C05446=1127.597,405.977,-90.668,-176.772,11.513,149.514
C05447=1127.600,405.729,-90.630,-176.772,11.509,149.513
C05448=1127.605,405.482,-90.592,-176.773,11.506,149.513
C05449=1127.608,405.235,-90.554,-176.773,11.502,149.512
C05450=1127.611,404.988,-90.515,-176.773,11.498,149.511
C05451=1127.615,404.742,-90.477,-176.773,11.494,149.510
C05452=1127.619,404.494,-90.439,-176.774,11.491,149.509
C05453=1127.622,404.247,-90.401,-176.773,11.488,149.508
C05454=1127.626,404.000,-90.362,-176.774,11.484,149.507
C05455=1127.630,403.753,-90.324,-176.774,11.481,149.506
C05456=1127.633,403.541,-90.291,-176.774,11.477,149.505
C05457=1127.637,403.328,-90.259,-176.774,11.474,149.505
C05458=1127.639,403.116,-90.225,-176.774,11.472,149.504
C05459=1127.643,402.904,-90.192,-176.775,11.468,149.503
C05460=1127.646,402.691,-90.160,-176.775,11.466,149.503
C05461=1127.649,402.480,-90.127,-176.775,11.462,149.502
C05462=1127.651,402.267,-90.094,-176.775,11.460,149.501
C05463=1127.655,402.055,-90.062,-176.776,11.457,149.501
C05464=1127.659,401.808,-90.023,-176.776,11.454,149.500
C05465=1127.662,401.561,-89.985,-176.777,11.450,149.499
C05466=1127.666,401.314,-89.947,-176.777,11.447,149.498
C05467=1127.670,401.067,-89.909,-176.778,11.443,149.498
C05468=1127.673,400.820,-89.871,-176.778,11.441,149.497
C05469=1127.677,400.572,-89.832,-176.778,11.437,149.496
C05470=1127.681,400.325,-89.795,-176.779,11.434,149.495
C05471=1127.684,400.078,-89.757,-176.779,11.431,149.495
C05472=1127.688,399.832,-89.718,-176.780,11.428,149.494
C05473=1127.692,399.585,-89.680,-176.781,11.425,149.493
C05474=1127.695,399.337,-89.641,-176.781,11.422,149.493
C05475=1127.699,399.091,-89.604,-176.781,11.419,149.492
C05476=1127.702,398.843,-89.566,-176.782,11.415,149.491
C05477=1127.707,398.596,-89.528,-176.782,11.413,149.491
C05478=1127.710,398.349,-89.490,-176.783,11.410,149.490
C05479=1127.714,398.102,-89.451,-176.784,11.407,149.490
C05480=1127.718,397.855,-89.414,-176.784,11.404,149.489
C05481=1127.721,397.608,-89.376,-176.785,11.401,149.488
C05482=1127.726,397.361,-89.338,-176.786,11.398,149.488
C05483=1127.729,397.114,-89.300,-176.787,11.396,149.487
C05484=1127.733,396.867,-89.262,-176.787,11.392,149.487
C05485=1127.736,396.619,-89.223,-176.788,11.389,149.486
C05486=1127.740,396.372,-89.186,-176.789,11.387,149.486
C05487=1127.743,396.126,-89.148,-176.790,11.384,149.485
C05488=1127.747,395.878,-89.109,-176.790,11.382,149.485
C05489=1127.751,395.631,-89.072,-176.791,11.379,149.484
C05490=1127.754,395.384,-89.034,-176.792,11.376,149.484
C05491=1127.759,395.137,-88.996,-176.793,11.373,149.483
C05492=1127.762,394.890,-88.958,-176.794,11.370,149.483
C05493=1127.766,394.643,-88.920,-176.795,11.368,149.482
C05494=1127.770,394.396,-88.882,-176.796,11.365,149.482
C05495=1127.773,394.149,-88.844,-176.796,11.363,149.481
C05496=1127.777,393.902,-88.806,-176.797,11.360,149.481
C05497=1127.780,393.655,-88.768,-176.798,11.358,149.481
C05498=1127.784,393.408,-88.730,-176.799,11.355,149.480
C05499=1127.788,393.161,-88.692,-176.800,11.353,149.480
C05500=1127.791,392.914,-88.655,-176.801,11.350,149.479
C05501=1127.796,392.666,-88.617,-176.802,11.348,149.479
C05502=1127.799,392.419,-88.579,-176.803,11.345,149.479
C05503=1127.803,392.172,-88.541,-176.804,11.343,149.478
C05504=1127.806,391.925,-88.504,-176.805,11.340,149.478
C05505=1127.810,391.678,-88.466,-176.806,11.339,149.477
C05506=1127.814,391.431,-88.428,-176.807,11.336,149.477
C05507=1127.817,391.184,-88.390,-176.808,11.334,149.477
C05508=1127.821,390.937,-88.352,-176.810,11.331,149.477
C05509=1127.825,390.689,-88.315,-176.811,11.329,149.476
C05510=1127.829,390.443,-88.277,-176.811,11.327,149.476
C05511=1127.832,390.195,-88.239,-176.813,11.325,149.476
C05512=1127.836,389.983,-88.206,-176.814,11.323,149.475
C05513=1127.839,389.771,-88.174,-176.815,11.321,149.475
C05514=1127.842,389.559,-88.142,-176.815,11.319,149.475
C05515=1127.845,389.346,-88.109,-176.817,11.318,149.475
C05516=1127.848,389.134,-88.077,-176.818,11.316,149.475
C05517=1127.851,388.921,-88.044,-176.818,11.314,149.474
C05518=1127.855,388.709,-88.011,-176.820,11.312,149.474
C05519=1127.857,388.497,-87.979,-176.821,11.309,149.474
C05520=1127.862,388.249,-87.942,-176.822,11.308,149.474
C05521=1127.865,388.002,-87.904,-176.823,11.306,149.473
C05522=1127.869,387.755,-87.866,-176.825,11.304,149.473
C05523=1127.872,387.508,-87.829,-176.826,11.302,149.473
C05524=1127.876,387.260,-87.791,-176.827,11.300,149.473
C05525=1127.880,387.014,-87.754,-176.829,11.297,149.473
C05526=1127.884,386.766,-87.715,-176.830,11.296,149.473
C05527=1127.888,386.519,-87.678,-176.832,11.294,149.472
C05528=1127.891,386.272,-87.640,-176.833,11.292,149.472
C05529=1127.895,386.025,-87.603,-176.834,11.290,149.472
C05530=1127.898,385.779,-87.565,-176.836,11.288,149.472
C05531=1127.902,385.531,-87.528,-176.837,11.286,149.472
C05532=1127.906,385.284,-87.490,-176.838,11.285,149.472
C05533=1127.909,385.037,-87.452,-176.840,11.282,149.472
C05534=1127.914,384.789,-87.415,-176.841,11.281,149.472
C05535=1127.917,384.542,-87.377,-176.843,11.279,149.471
C05536=1127.921,384.295,-87.340,-176.845,11.277,149.471
C05537=1127.924,384.048,-87.302,-176.846,11.275,149.471
C05538=1127.928,383.801,-87.265,-176.847,11.274,149.471
C05539=1127.932,383.554,-87.228,-176.849,11.271,149.471
C05540=1127.935,383.307,-87.190,-176.851,11.269,149.471
C05541=1127.939,383.060,-87.152,-176.853,11.267,149.471
C05542=1127.943,382.812,-87.115,-176.856,11.264,149.471
C05543=1127.946,382.566,-87.078,-176.859,11.262,149.471
C05544=1127.951,382.318,-87.040,-176.862,11.260,149.471
C05545=1127.954,382.071,-87.002,-176.865,11.257,149.471
C05546=1127.958,381.824,-86.965,-176.867,11.255,149.471
C05547=1127.962,381.576,-86.927,-176.870,11.252,149.472
C05548=1127.966,381.329,-86.891,-176.873,11.250,149.472
C05549=1127.969,381.083,-86.853,-176.876,11.248,149.472
C05550=1127.973,380.835,-86.816,-176.878,11.246,149.472
C05551=1127.977,380.588,-86.778,-176.881,11.243,149.472
C05552=1127.980,380.340,-86.741,-176.884,11.240,149.472
C05553=1127.984,380.094,-86.703,-176.887,11.239,149.472
C05554=1127.988,379.846,-86.666,-176.890,11.236,149.472
C05555=1127.992,379.599,-86.629,-176.892,11.233,149.472
C05556=1127.995,379.352,-86.592,-176.895,11.231,149.472
C05557=1128.000,379.105,-86.555,-176.898,11.228,149.472
C05558=1128.003,378.858,-86.517,-176.901,11.227,149.473
C05559=1128.007,378.610,-86.480,-176.904,11.224,149.473
C05560=1128.011,378.363,-86.443,-176.907,11.221,149.473
C05561=1128.013,378.116,-86.406,-176.909,11.219,149.473
C05562=1128.017,377.869,-86.369,-176.912,11.217,149.473
C05563=1128.022,377.622,-86.332,-176.915,11.214,149.473
C05564=1128.025,377.374,-86.295,-176.918,11.212,149.473
C05565=1128.029,377.127,-86.257,-176.921,11.210,149.474
C05566=1128.033,376.880,-86.220,-176.924,11.208,149.474
C05567=1128.037,376.633,-86.184,-176.927,11.205,149.474
C05568=1128.040,376.421,-86.152,-176.929,11.203,149.474
C05569=1128.044,376.208,-86.120,-176.932,11.202,149.474
C05570=1128.046,375.996,-86.088,-176.935,11.199,149.474
C05571=1128.050,375.783,-86.056,-176.937,11.197,149.474
C05572=1128.053,375.570,-86.025,-176.940,11.195,149.475
C05573=1128.056,375.358,-85.993,-176.942,11.193,149.475
C05574=1128.060,375.145,-85.961,-176.945,11.191,149.475
C05575=1128.062,374.933,-85.929,-176.947,11.189,149.475
C05576=1128.066,374.685,-85.892,-176.950,11.187,149.475
C05577=1128.070,374.438,-85.855,-176.954,11.184,149.475
C05578=1128.074,374.191,-85.818,-176.956,11.183,149.476
C05579=1128.077,373.944,-85.782,-176.959,11.180,149.476
C05580=1128.081,373.696,-85.744,-176.962,11.178,149.476
C05581=1128.085,373.449,-85.707,-176.966,11.175,149.476
C05582=1128.089,373.202,-85.671,-176.968,11.173,149.476
C05583=1128.093,372.955,-85.634,-176.972,11.171,149.476
C05584=1128.097,372.708,-85.597,-176.975,11.168,149.477
C05585=1128.100,372.460,-85.560,-176.977,11.166,149.477
C05586=1128.104,372.213,-85.523,-176.981,11.164,149.477
C05587=1128.107,371.966,-85.487,-176.984,11.161,149.477
C05588=1128.112,371.719,-85.450,-176.987,11.159,149.477
C05589=1128.116,371.471,-85.413,-176.990,11.157,149.478
C05590=1128.119,371.224,-85.376,-176.993,11.155,149.478
C05591=1128.123,370.977,-85.340,-176.996,11.152,149.478
C05592=1128.127,370.729,-85.303,-177.000,11.150,149.478
C05593=1128.131,370.482,-85.266,-177.002,11.148,149.478
C05594=1128.134,370.235,-85.230,-177.006,11.146,149.479
C05595=1128.138,369.988,-85.193,-177.009,11.143,149.479
C05596=1128.142,369.740,-85.156,-177.012,11.141,149.479
C05597=1128.145,369.493,-85.120,-177.016,11.138,149.479
C05598=1128.149,369.246,-85.083,-177.018,11.137,149.480
C05599=1128.154,368.998,-85.047,-177.022,11.134,149.480
C05600=1128.157,368.752,-85.010,-177.025,11.132,149.480
C05601=1128.161,368.504,-84.973,-177.028,11.129,149.480
C05602=1128.164,368.258,-84.937,-177.031,11.127,149.480
C05603=1128.168,368.009,-84.901,-177.034,11.125,149.481
C05604=1128.172,367.762,-84.864,-177.037,11.122,149.481
C05605=1128.176,367.515,-84.828,-177.041,11.120,149.481
C05606=1128.180,367.267,-84.791,-177.044,11.117,149.481
C05607=1128.183,367.020,-84.755,-177.047,11.115,149.481
C05608=1128.187,366.773,-84.718,-177.051,11.113,149.482
C05609=1128.191,366.526,-84.682,-177.054,11.110,149.482
C05610=1128.195,366.278,-84.646,-177.057,11.108,149.482
C05611=1128.199,366.031,-84.610,-177.060,11.106,149.483
C05612=1128.203,365.784,-84.573,-177.064,11.104,149.483
C05613=1128.207,365.536,-84.537,-177.067,11.101,149.483
C05614=1128.210,365.289,-84.500,-177.070,11.099,149.483
C05615=1128.214,365.041,-84.464,-177.073,11.096,149.483
C05616=1128.218,364.794,-84.428,-177.077,11.094,149.484
C05617=1128.221,364.547,-84.392,-177.080,11.091,149.484
C05618=1128.225,364.299,-84.355,-177.084,11.089,149.484
C05619=1128.229,364.053,-84.319,-177.086,11.088,149.484
C05620=1128.233,363.805,-84.283,-177.090,11.085,149.485
C05621=1128.236,363.558,-84.247,-177.093,11.083,149.485
C05622=1128.241,363.310,-84.210,-177.096,11.080,149.485
C05623=1128.244,363.063,-84.174,-177.100,11.078,149.485
C05624=1128.248,362.850,-84.144,-177.103,11.075,149.486
C05625=1128.251,362.637,-84.112,-177.106,11.074,149.486
C05626=1128.254,362.425,-84.081,-177.108,11.072,149.486
C05627=1128.257,362.213,-84.050,-177.112,11.069,149.486
C05628=1128.261,361.999,-84.020,-177.114,11.068,149.486
C05629=1128.264,361.787,-83.988,-177.118,11.065,149.487
C05630=1128.267,361.575,-83.957,-177.120,11.064,149.487
C05631=1128.271,361.362,-83.927,-177.124,11.061,149.487
C05632=1128.274,361.115,-83.891,-177.127,11.059,149.487
C05633=1128.278,360.867,-83.854,-177.130,11.056,149.488
C05634=1128.282,360.619,-83.819,-177.134,11.054,149.488
C05635=1128.285,360.372,-83.783,-177.137,11.052,149.488
C05636=1128.290,360.125,-83.746,-177.141,11.049,149.488
C05637=1128.293,359.877,-83.711,-177.144,11.047,149.489
C05638=1128.297,359.630,-83.675,-177.147,11.044,149.489
C05639=1128.301,359.382,-83.638,-177.151,11.042,149.489
C05640=1128.305,359.135,-83.603,-177.154,11.039,149.490
C05641=1128.309,358.887,-83.567,-177.157,11.037,149.490
C05642=1128.312,358.641,-83.531,-177.161,11.035,149.490
C05643=1128.316,358.393,-83.495,-177.164,11.032,149.490
C05644=1128.321,358.146,-83.460,-177.168,11.030,149.491
C05645=1128.324,357.898,-83.424,-177.171,11.027,149.491
C05646=1128.328,357.651,-83.389,-177.174,11.025,149.491
C05647=1128.332,357.403,-83.353,-177.178,11.023,149.491
C05648=1128.336,357.156,-83.317,-177.182,11.020,149.492
C05649=1128.339,356.909,-83.281,-177.185,11.017,149.492
C05650=1128.343,356.661,-83.245,-177.189,11.015,149.492
C05651=1128.347,356.414,-83.210,-177.192,11.013,149.492
C05652=1128.350,356.166,-83.174,-177.196,11.010,149.493
C05653=1128.355,355.920,-83.139,-177.199,11.008,149.493
C05654=1128.359,355.672,-83.103,-177.203,11.005,149.493
C05655=1128.363,355.424,-83.067,-177.207,11.002,149.493
C05656=1128.366,355.177,-83.032,-177.210,11.000,149.494
C05657=1128.370,354.929,-82.996,-177.213,10.997,149.494
C05658=1128.374,354.682,-82.961,-177.217,10.995,149.494
C05659=1128.378,354.435,-82.925,-177.221,10.992,149.495
C05660=1128.382,354.187,-82.890,-177.224,10.989,149.495
C05661=1128.385,353.940,-82.854,-177.228,10.987,149.495
C05662=1128.389,353.692,-82.819,-177.231,10.985,149.495
C05663=1128.394,353.444,-82.783,-177.235,10.982,149.496
C05664=1128.398,353.197,-82.748,-177.238,10.979,149.496
C05665=1128.402,352.950,-82.713,-177.242,10.977,149.496
C05666=1128.405,352.702,-82.677,-177.245,10.975,149.496
C05667=1128.409,352.455,-82.642,-177.249,10.971,149.497
C05668=1128.413,352.208,-82.606,-177.253,10.969,149.497
C05669=1128.417,351.960,-82.571,-177.256,10.966,149.497
C05670=1128.421,351.712,-82.536,-177.260,10.964,149.497
C05671=1128.424,351.465,-82.500,-177.264,10.961,149.498
C05672=1128.429,351.218,-82.465,-177.267,10.959,149.498
C05673=1128.433,350.970,-82.430,-177.271,10.955,149.498
C05674=1128.436,350.722,-82.395,-177.275,10.953,149.498
C05675=1128.440,350.475,-82.359,-177.278,10.951,149.499
C05676=1128.444,350.228,-82.325,-177.282,10.948,149.499
C05677=1128.447,349.980,-82.290,-177.285,10.945,149.499
C05678=1128.451,349.733,-82.254,-177.289,10.943,149.500
C05679=1128.456,349.485,-82.220,-177.293,10.940,149.500
C05680=1128.459,349.272,-82.189,-177.295,10.938,149.500
C05681=1128.463,349.059,-82.159,-177.298,10.935,149.500
C05682=1128.466,348.846,-82.129,-177.301,10.934,149.500
C05683=1128.469,348.633,-82.099,-177.303,10.932,149.500
C05684=1128.472,348.421,-82.069,-177.307,10.929,149.501
C05685=1128.476,348.208,-82.038,-177.309,10.927,149.501
C05686=1128.479,347.995,-82.008,-177.312,10.925,149.501
C05687=1128.482,347.782,-81.978,-177.315,10.923,149.501
C05688=1128.486,347.535,-81.943,-177.318,10.920,149.501
C05689=1128.490,347.287,-81.908,-177.321,10.918,149.501
C05690=1128.494,347.040,-81.873,-177.325,10.915,149.502
C05691=1128.499,346.792,-81.838,-177.328,10.913,149.502
C05692=1128.502,346.544,-81.804,-177.331,10.910,149.502
C05693=1128.506,346.298,-81.769,-177.335,10.908,149.502
C05694=1128.510,346.050,-81.734,-177.338,10.905,149.503
C05695=1128.514,345.802,-81.698,-177.341,10.903,149.503
C05696=1128.518,345.555,-81.664,-177.344,10.900,149.503
C05697=1128.521,345.307,-81.630,-177.347,10.898,149.503
C05698=1128.526,345.060,-81.595,-177.351,10.895,149.503
C05699=1128.530,344.812,-81.560,-177.354,10.893,149.504
C05700=1128.534,344.564,-81.525,-177.357,10.890,149.504
C05701=1128.537,344.317,-81.490,-177.360,10.889,149.504
C05702=1128.541,344.069,-81.455,-177.363,10.886,149.504
C05703=1128.546,343.822,-81.421,-177.366,10.883,149.504
C05704=1128.549,343.575,-81.386,-177.370,10.881,149.505
C05705=1128.553,343.327,-81.352,-177.373,10.878,149.505
C05706=1128.557,343.079,-81.317,-177.376,10.876,149.505
C05707=1128.562,342.832,-81.282,-177.379,10.874,149.505
C05708=1128.565,342.584,-81.247,-177.383,10.871,149.506
C05709=1128.569,342.336,-81.212,-177.386,10.868,149.506
C05710=1128.573,342.089,-81.178,-177.389,10.866,149.506
C05711=1128.576,341.841,-81.144,-177.392,10.863,149.506
C05712=1128.581,341.594,-81.109,-177.396,10.861,149.506
C05713=1128.584,341.346,-81.075,-177.399,10.859,149.507
C05714=1128.589,341.099,-81.040,-177.402,10.856,149.507
C05715=1128.593,340.851,-81.005,-177.405,10.853,149.507
C05716=1128.596,340.604,-80.971,-177.409,10.851,149.507
C05717=1128.601,340.356,-80.937,-177.412,10.848,149.507
C05718=1128.605,340.108,-80.902,-177.415,10.846,149.507
C05719=1128.609,339.861,-80.868,-177.418,10.843,149.508
C05720=1128.613,339.613,-80.833,-177.421,10.841,149.508
C05721=1128.617,339.366,-80.799,-177.425,10.838,149.508
C05722=1128.620,339.118,-80.764,-177.428,10.836,149.508
C05723=1128.624,338.871,-80.731,-177.431,10.833,149.508
C05724=1128.628,338.623,-80.696,-177.434,10.831,149.509
C05725=1128.632,338.375,-80.662,-177.438,10.828,149.509
C05726=1128.636,338.127,-80.627,-177.440,10.826,149.509
C05727=1128.640,337.880,-80.593,-177.444,10.824,149.509
C05728=1128.644,337.633,-80.559,-177.447,10.822,149.510
C05729=1128.648,337.385,-80.525,-177.450,10.819,149.510
C05730=1128.652,337.138,-80.490,-177.453,10.816,149.510
C05731=1128.656,336.890,-80.456,-177.456,10.814,149.510
C05732=1128.660,336.642,-80.422,-177.460,10.811,149.510
C05733=1128.664,336.394,-80.388,-177.463,10.809,149.511
C05734=1128.668,336.147,-80.353,-177.466,10.806,149.511
C05735=1128.672,335.899,-80.319,-177.469,10.804,149.511
C05736=1128.675,335.686,-80.290,-177.472,10.802,149.511
C05737=1128.679,335.473,-80.260,-177.475,10.799,149.511
C05738=1128.682,335.260,-80.231,-177.478,10.798,149.511
C05739=1128.685,335.047,-80.202,-177.481,10.795,149.511
C05740=1128.689,334.834,-80.173,-177.483,10.793,149.512
C05741=1128.692,334.622,-80.143,-177.486,10.790,149.512
C05742=1128.696,334.409,-80.115,-177.489,10.789,149.512
C05743=1128.699,334.195,-80.085,-177.491,10.787,149.512
C05744=1128.703,333.948,-80.051,-177.494,10.784,149.512
C05745=1128.707,333.701,-80.017,-177.498,10.782,149.513
C05746=1128.711,333.452,-79.983,-177.501,10.779,149.513
C05747=1128.715,333.205,-79.949,-177.504,10.776,149.513
C05748=1128.719,332.958,-79.915,-177.507,10.774,149.513
C05749=1128.723,332.709,-79.881,-177.511,10.772,149.513
C05750=1128.727,332.462,-79.847,-177.514,10.769,149.513
C05751=1128.731,332.214,-79.814,-177.517,10.766,149.514
C05752=1128.735,331.966,-79.779,-177.520,10.764,149.514
C05753=1128.739,331.719,-79.745,-177.524,10.761,149.514
C05754=1128.743,331.471,-79.712,-177.526,10.759,149.514
C05755=1128.746,331.223,-79.678,-177.530,10.756,149.514
C05756=1128.751,330.975,-79.644,-177.533,10.754,149.515
C05757=1128.755,330.728,-79.610,-177.536,10.751,149.515
C05758=1128.759,330.480,-79.577,-177.539,10.749,149.515
C05759=1128.762,330.233,-79.543,-177.543,10.746,149.515
C05760=1128.766,329.985,-79.510,-177.546,10.744,149.516
C05761=1128.771,329.737,-79.475,-177.548,10.742,149.516
C05762=1128.775,329.489,-79.442,-177.552,10.739,149.516
C05763=1128.778,329.242,-79.408,-177.555,10.737,149.516
C05764=1128.783,328.994,-79.375,-177.558,10.734,149.516
C05765=1128.786,328.747,-79.341,-177.561,10.732,149.516
C05766=1128.791,328.498,-79.307,-177.564,10.729,149.517
C05767=1128.795,328.251,-79.274,-177.568,10.727,149.517
C05768=1128.799,328.004,-79.240,-177.571,10.724,149.517
C05769=1128.803,327.756,-79.206,-177.574,10.721,149.517
C05770=1128.807,327.508,-79.173,-177.577,10.719,149.517
C05771=1128.810,327.260,-79.139,-177.581,10.717,149.518
C05772=1128.814,327.013,-79.106,-177.584,10.714,149.518
C05773=1128.818,326.765,-79.073,-177.587,10.711,149.518
C05774=1128.823,326.517,-79.038,-177.590,10.709,149.518
C05775=1128.827,326.270,-79.005,-177.593,10.706,149.518
C05776=1128.831,326.021,-78.972,-177.597,10.704,149.519
C05777=1128.835,325.773,-78.938,-177.600,10.701,149.519
C05778=1128.839,325.526,-78.905,-177.603,10.698,149.519
C05779=1128.843,325.279,-78.871,-177.606,10.696,149.519
C05780=1128.847,325.031,-78.838,-177.609,10.694,149.519
C05781=1128.851,324.783,-78.805,-177.612,10.691,149.519
C05782=1128.855,324.535,-78.772,-177.615,10.689,149.520
C05783=1128.858,324.288,-78.738,-177.618,10.687,149.520
C05784=1128.863,324.040,-78.705,-177.622,10.684,149.520
C05785=1128.867,323.792,-78.671,-177.625,10.681,149.520
C05786=1128.871,323.544,-78.638,-177.628,10.679,149.521
C05787=1128.875,323.297,-78.605,-177.631,10.677,149.521
C05788=1128.879,323.049,-78.572,-177.634,10.674,149.521
C05789=1128.883,322.801,-78.539,-177.637,10.671,149.521
C05790=1128.887,322.553,-78.505,-177.641,10.669,149.521
C05791=1128.891,322.305,-78.472,-177.644,10.666,149.521
C05792=1128.894,322.093,-78.444,-177.646,10.664,149.522
C05793=1128.898,321.879,-78.416,-177.649,10.662,149.522
C05794=1128.901,321.666,-78.387,-177.652,10.660,149.522
C05795=1128.905,321.453,-78.358,-177.655,10.657,149.522
C05796=1128.908,321.240,-78.330,-177.657,10.655,149.522
C05797=1128.911,321.027,-78.301,-177.660,10.654,149.522
C05798=1128.915,320.814,-78.273,-177.663,10.651,149.523
C05799=1128.919,320.601,-78.244,-177.666,10.649,149.523
C05800=1128.923,320.353,-78.211,-177.669,10.646,149.523
C05801=1128.927,320.105,-78.178,-177.672,10.644,149.523
C05802=1128.930,319.857,-78.145,-177.675,10.641,149.523
C05803=1128.934,319.610,-78.112,-177.678,10.639,149.523
C05804=1128.938,319.361,-78.080,-177.681,10.636,149.524
C05805=1128.942,319.113,-78.046,-177.684,10.633,149.524
C05806=1128.946,318.866,-78.013,-177.688,10.631,149.524
C05807=1128.950,318.618,-77.981,-177.691,10.629,149.524
C05808=1128.954,318.371,-77.948,-177.694,10.626,149.524
C05809=1128.958,318.123,-77.914,-177.697,10.623,149.525
C05810=1128.963,317.874,-77.882,-177.701,10.621,149.525
C05811=1128.967,317.627,-77.849,-177.703,10.619,149.525
C05812=1128.970,317.379,-77.816,-177.706,10.617,149.525
C05813=1128.974,317.132,-77.783,-177.710,10.614,149.525
C05814=1128.979,316.883,-77.751,-177.712,10.611,149.526
C05815=1128.983,316.636,-77.717,-177.716,10.609,149.526
C05816=1128.986,316.388,-77.685,-177.719,10.606,149.526
C05817=1128.991,316.140,-77.652,-177.722,10.604,149.526
C05818=1128.995,315.892,-77.619,-177.725,10.601,149.526
C05819=1128.998,315.645,-77.587,-177.728,10.598,149.526
C05820=1129.003,315.396,-77.554,-177.732,10.596,149.527
C05821=1129.007,315.149,-77.522,-177.735,10.593,149.527
C05822=1129.011,314.902,-77.489,-177.738,10.591,149.527
C05823=1129.015,314.653,-77.457,-177.741,10.588,149.527
C05824=1129.019,314.406,-77.423,-177.744,10.586,149.527
C05825=1129.023,314.158,-77.392,-177.747,10.583,149.528
C05826=1129.027,313.910,-77.358,-177.750,10.580,149.528
C05827=1129.031,313.662,-77.325,-177.754,10.578,149.528
C05828=1129.035,313.414,-77.293,-177.757,10.575,149.528
C05829=1129.039,313.166,-77.260,-177.759,10.573,149.528
C05830=1129.043,312.918,-77.228,-177.763,10.571,149.529
C05831=1129.047,312.671,-77.195,-177.766,10.568,149.529
C05832=1129.052,312.422,-77.163,-177.769,10.566,149.529
C05833=1129.056,312.176,-77.131,-177.772,10.563,149.529
C05834=1129.060,311.927,-77.098,-177.775,10.561,149.529
C05835=1129.064,311.679,-77.066,-177.779,10.558,149.529
C05836=1129.068,311.432,-77.033,-177.781,10.555,149.530
C05837=1129.072,311.183,-77.001,-177.785,10.553,149.530
C05838=1129.076,310.936,-76.968,-177.788,10.551,149.530
C05839=1129.079,310.688,-76.936,-177.791,10.548,149.530
C05840=1129.084,310.440,-76.904,-177.794,10.545,149.530
C05841=1129.088,310.193,-76.872,-177.797,10.543,149.530
C05842=1129.092,309.944,-76.839,-177.801,10.540,149.531
C05843=1129.096,309.696,-76.807,-177.804,10.537,149.531
C05844=1129.100,309.449,-76.774,-177.807,10.535,149.531
C05845=1129.104,309.200,-76.742,-177.810,10.533,149.531
C05846=1129.109,308.953,-76.710,-177.813,10.531,149.531
C05847=1129.113,308.705,-76.678,-177.816,10.528,149.532
C05848=1129.116,308.491,-76.650,-177.819,10.525,149.532
C05849=1129.119,308.278,-76.623,-177.821,10.523,149.532
C05850=1129.123,308.065,-76.595,-177.824,10.522,149.532
C05851=1129.126,307.851,-76.567,-177.827,10.519,149.532
C05852=1129.130,307.639,-76.540,-177.829,10.517,149.533
C05853=1129.134,307.425,-76.512,-177.832,10.514,149.533
C05854=1129.137,307.212,-76.484,-177.835,10.512,149.533
C05855=1129.141,306.998,-76.457,-177.837,10.511,149.533
C05856=1129.145,306.751,-76.424,-177.840,10.508,149.533
C05857=1129.149,306.503,-76.393,-177.844,10.506,149.533
C05858=1129.153,306.255,-76.360,-177.847,10.503,149.533
C05859=1129.157,306.007,-76.328,-177.850,10.500,149.534
C05860=1129.161,305.759,-76.296,-177.853,10.498,149.534
C05861=1129.166,305.511,-76.264,-177.856,10.495,149.534
C05862=1129.169,305.263,-76.232,-177.859,10.492,149.534
C05863=1129.174,305.015,-76.200,-177.862,10.490,149.534
C05864=1129.178,304.768,-76.169,-177.865,10.487,149.534
C05865=1129.182,304.519,-76.137,-177.869,10.485,149.535
C05866=1129.186,304.271,-76.105,-177.872,10.482,149.535
C05867=1129.190,304.023,-76.072,-177.875,10.480,149.535
C05868=1129.194,303.776,-76.041,-177.878,10.478,149.535
C05869=1129.198,303.528,-76.009,-177.881,10.475,149.535
C05870=1129.203,303.279,-75.977,-177.884,10.473,149.536
C05871=1129.207,303.032,-75.945,-177.887,10.470,149.536
C05872=1129.211,302.784,-75.913,-177.890,10.468,149.536
C05873=1129.214,302.536,-75.881,-177.893,10.465,149.536
C05874=1129.219,302.288,-75.849,-177.896,10.462,149.536
C05875=1129.223,302.040,-75.818,-177.899,10.460,149.536
C05876=1129.227,301.793,-75.786,-177.903,10.457,149.537
C05877=1129.231,301.544,-75.755,-177.906,10.454,149.537
C05878=1129.235,301.296,-75.723,-177.909,10.452,149.537
C05879=1129.240,301.049,-75.691,-177.912,10.449,149.537
C05880=1129.244,300.801,-75.659,-177.915,10.447,149.537
C05881=1129.247,300.552,-75.627,-177.919,10.444,149.538
C05882=1129.252,300.305,-75.597,-177.921,10.442,149.538
C05883=1129.256,300.056,-75.565,-177.924,10.440,149.538
C05884=1129.260,299.809,-75.533,-177.927,10.437,149.538
C05885=1129.265,299.561,-75.501,-177.930,10.435,149.538
C05886=1129.269,299.312,-75.470,-177.933,10.432,149.538
C05887=1129.273,299.065,-75.438,-177.937,10.430,149.539
C05888=1129.277,298.817,-75.406,-177.940,10.427,149.539
C05889=1129.281,298.569,-75.376,-177.943,10.424,149.539
C05890=1129.285,298.321,-75.344,-177.946,10.422,149.539
C05891=1129.289,298.073,-75.312,-177.949,10.419,149.539
C05892=1129.293,297.825,-75.281,-177.952,10.416,149.540
C05893=1129.297,297.577,-75.249,-177.956,10.414,149.540
C05894=1129.301,297.329,-75.218,-177.958,10.411,149.540
C05895=1129.305,297.081,-75.187,-177.961,10.410,149.540
C05896=1129.310,296.833,-75.155,-177.964,10.407,149.540
C05897=1129.314,296.585,-75.124,-177.967,10.404,149.541
C05898=1129.318,296.337,-75.093,-177.970,10.402,149.541
C05899=1129.322,296.089,-75.060,-177.974,10.399,149.541
C05900=1129.326,295.841,-75.030,-177.977,10.396,149.541
C05901=1129.330,295.593,-74.998,-177.980,10.394,149.541
C05902=1129.334,295.345,-74.967,-177.983,10.391,149.541
C05903=1129.338,295.097,-74.936,-177.986,10.389,149.542
C05904=1129.342,294.884,-74.909,-177.989,10.387,149.542
C05905=1129.346,294.670,-74.882,-177.991,10.384,149.542
C05906=1129.349,294.457,-74.855,-177.994,10.382,149.542
C05907=1129.352,294.243,-74.828,-177.996,10.380,149.542
C05908=1129.356,294.030,-74.801,-177.999,10.378,149.542
C05909=1129.359,293.817,-74.774,-178.002,10.376,149.542
C05910=1129.363,293.603,-74.748,-178.004,10.374,149.543
C05911=1129.367,293.390,-74.721,-178.007,10.371,149.543
C05912=1129.371,293.142,-74.689,-178.010,10.368,149.543
C05913=1129.375,292.894,-74.658,-178.014,10.366,149.543
C05914=1129.380,292.646,-74.628,-178.017,10.363,149.543
C05915=1129.384,292.398,-74.596,-178.019,10.362,149.544
C05916=1129.388,292.150,-74.565,-178.022,10.359,149.544
C05917=1129.391,291.901,-74.535,-178.026,10.356,149.544
C05918=1129.396,291.653,-74.504,-178.028,10.354,149.544
C05919=1129.400,291.405,-74.472,-178.032,10.351,149.544
C05920=1129.404,291.157,-74.441,-178.035,10.348,149.544
C05921=1129.408,290.909,-74.410,-178.038,10.346,149.544
C05922=1129.413,290.661,-74.379,-178.041,10.343,149.545
C05923=1129.417,290.414,-74.348,-178.044,10.341,149.545
C05924=1129.421,290.165,-74.317,-178.047,10.338,149.545
C05925=1129.425,289.917,-74.286,-178.050,10.335,149.545
C05926=1129.429,289.668,-74.255,-178.054,10.333,149.545
C05927=1129.433,289.421,-74.224,-178.056,10.331,149.546
C05928=1129.437,289.173,-74.194,-178.059,10.329,149.546
C05929=1129.441,288.925,-74.163,-178.062,10.326,149.546
C05930=1129.446,288.677,-74.132,-178.066,10.323,149.546
C05931=1129.450,288.429,-74.102,-178.068,10.321,149.546
C05932=1129.454,288.180,-74.071,-178.071,10.318,149.546
C05933=1129.458,287.933,-74.040,-178.075,10.315,149.547
C05934=1129.463,287.685,-74.009,-178.078,10.313,149.547
C05935=1129.466,287.436,-73.978,-178.081,10.310,149.547
C05936=1129.471,287.188,-73.948,-178.084,10.307,149.547
C05937=1129.476,286.940,-73.917,-178.087,10.305,149.547
C05938=1129.479,286.692,-73.886,-178.090,10.303,149.548
C05939=1129.483,286.444,-73.856,-178.093,10.301,149.548
C05940=1129.488,286.196,-73.825,-178.096,10.298,149.548
C05941=1129.491,285.948,-73.794,-178.099,10.295,149.548
C05942=1129.496,285.700,-73.764,-178.102,10.293,149.548
C05943=1129.501,285.452,-73.733,-178.105,10.290,149.548
C05944=1129.504,285.203,-73.702,-178.108,10.288,149.549
C05945=1129.508,284.955,-73.672,-178.111,10.285,149.549
C05946=1129.512,284.708,-73.641,-178.115,10.282,149.549
C05947=1129.517,284.460,-73.611,-178.118,10.280,149.549
C05948=1129.521,284.211,-73.579,-178.120,10.278,149.549
C05949=1129.525,283.964,-73.549,-178.123,10.275,149.550
C05950=1129.530,283.715,-73.519,-178.126,10.272,149.550
C05951=1129.534,283.467,-73.489,-178.130,10.270,149.550
C05952=1129.538,283.219,-73.458,-178.132,10.267,149.550
C05953=1129.542,282.971,-73.428,-178.136,10.265,149.550
C05954=1129.546,282.723,-73.397,-178.139,10.262,149.550
C05955=1129.550,282.475,-73.367,-178.142,10.260,149.551
C05956=1129.554,282.226,-73.336,-178.145,10.257,149.551
C05957=1129.558,281.979,-73.306,-178.148,10.254,149.551
C05958=1129.563,281.731,-73.275,-178.151,10.252,149.551
C05959=1129.567,281.482,-73.246,-178.154,10.250,149.551
C05960=1129.570,281.268,-73.219,-178.157,10.247,149.552
C05961=1129.574,281.055,-73.193,-178.160,10.245,149.552
C05962=1129.578,280.842,-73.167,-178.163,10.242,149.552
C05963=1129.581,280.628,-73.141,-178.166,10.239,149.552
C05964=1129.586,280.414,-73.115,-178.170,10.237,149.552
C05965=1129.588,280.201,-73.089,-178.172,10.235,149.552
C05966=1129.593,279.987,-73.063,-178.175,10.233,149.553
C05967=1129.596,279.774,-73.038,-178.178,10.230,149.553
C05968=1129.600,279.525,-73.007,-178.181,10.227,149.553
C05969=1129.604,279.277,-72.976,-178.185,10.224,149.553
C05970=1129.608,279.029,-72.947,-178.188,10.221,149.553
C05971=1129.613,278.781,-72.916,-178.192,10.218,149.554
C05972=1129.617,278.533,-72.887,-178.195,10.215,149.554
C05973=1129.622,278.285,-72.856,-178.199,10.213,149.554
C05974=1129.626,278.037,-72.826,-178.202,10.210,149.554
C05975=1129.629,277.788,-72.796,-178.206,10.207,149.554
C05976=1129.634,277.540,-72.766,-178.209,10.204,149.555
C05977=1129.638,277.292,-72.736,-178.212,10.202,149.555
C05978=1129.642,277.044,-72.706,-178.215,10.198,149.555
C05979=1129.646,276.796,-72.676,-178.219,10.196,149.555
C05980=1129.651,276.548,-72.646,-178.222,10.193,149.555
C05981=1129.655,276.299,-72.617,-178.225,10.190,149.555
C05982=1129.659,276.052,-72.586,-178.228,10.188,149.556
C05983=1129.663,275.803,-72.557,-178.231,10.185,149.556
C05984=1129.668,275.555,-72.526,-178.235,10.182,149.556
C05985=1129.671,275.307,-72.496,-178.238,10.179,149.556
C05986=1129.676,275.058,-72.467,-178.241,10.177,149.556
C05987=1129.679,274.811,-72.437,-178.244,10.174,149.556
C05988=1129.684,274.562,-72.407,-178.247,10.171,149.556
C05989=1129.688,274.314,-72.377,-178.250,10.169,149.557
C05990=1129.693,274.065,-72.348,-178.253,10.166,149.557
C05991=1129.697,273.818,-72.318,-178.256,10.163,149.557
C05992=1129.701,273.570,-72.288,-178.259,10.160,149.557
C05993=1129.706,273.321,-72.258,-178.262,10.158,149.557
C05994=1129.710,273.073,-72.229,-178.265,10.155,149.557
C05995=1129.714,272.825,-72.198,-178.268,10.152,149.558
C05996=1129.718,272.577,-72.169,-178.271,10.150,149.558
C05997=1129.722,272.329,-72.140,-178.274,10.147,149.558
C05998=1129.726,272.080,-72.110,-178.277,10.144,149.558
C05999=1129.730,271.832,-72.081,-178.280,10.141,149.558
C06000=1129.735,271.584,-72.051,-178.282,10.139,149.558
C06001=1129.740,271.335,-72.021,-178.285,10.137,149.558
C06002=1129.743,271.088,-71.991,-178.288,10.134,149.558
C06003=1129.748,270.839,-71.962,-178.291,10.131,149.558
C06004=1129.752,270.591,-71.932,-178.294,10.128,149.559
C06005=1129.756,270.343,-71.903,-178.296,10.126,149.559
C06006=1129.760,270.094,-71.873,-178.299,10.124,149.559
C06007=1129.764,269.846,-71.844,-178.302,10.121,149.559
C06008=1129.769,269.599,-71.815,-178.305,10.118,149.559
C06009=1129.773,269.350,-71.785,-178.307,10.116,149.559
C06010=1129.777,269.102,-71.756,-178.310,10.113,149.559
C06011=1129.782,268.854,-71.726,-178.313,10.111,149.559
C06012=1129.786,268.606,-71.697,-178.316,10.109,149.559
C06013=1129.790,268.357,-71.667,-178.318,10.106,149.560
C06014=1129.794,268.109,-71.638,-178.321,10.104,149.560
C06015=1129.798,267.861,-71.608,-178.324,10.101,149.560
C06016=1129.802,267.647,-71.583,-178.326,10.099,149.560
C06017=1129.807,267.433,-71.558,-178.328,10.097,149.560
C06018=1129.810,267.220,-71.533,-178.330,10.095,149.560
C06019=1129.813,267.005,-71.508,-178.333,10.093,149.560
C06020=1129.817,266.792,-71.482,-178.335,10.091,149.560
C06021=1129.820,266.579,-71.457,-178.337,10.089,149.560
C06022=1129.824,266.365,-71.433,-178.339,10.087,149.560
C06023=1129.828,266.151,-71.407,-178.341,10.085,149.560
C06024=1129.833,265.903,-71.377,-178.344,10.082,149.560
C06025=1129.837,265.654,-71.348,-178.346,10.080,149.560
C06026=1129.840,265.406,-71.319,-178.348,10.078,149.561
C06027=1129.844,265.158,-71.290,-178.351,10.075,149.561
C06028=1129.849,264.910,-71.261,-178.354,10.073,149.561
C06029=1129.854,264.662,-71.232,-178.356,10.071,149.561
C06030=1129.858,264.413,-71.202,-178.359,10.068,149.561
C06031=1129.862,264.165,-71.173,-178.363,10.065,149.561
C06032=1129.866,263.916,-71.144,-178.367,10.062,149.562
C06033=1129.871,263.668,-71.115,-178.371,10.058,149.562
C06034=1129.875,263.421,-71.086,-178.375,10.055,149.562
C06035=1129.879,263.172,-71.058,-178.378,10.053,149.562
C06036=1129.883,262.923,-71.028,-178.382,10.049,149.563
C06037=1129.888,262.675,-70.999,-178.385,10.046,149.563
C06038=1129.892,262.426,-70.970,-178.389,10.043,149.563
C06039=1129.897,262.179,-70.941,-178.393,10.040,149.563
C06040=1129.900,261.931,-70.912,-178.396,10.037,149.563
C06041=1129.905,261.682,-70.883,-178.400,10.034,149.564
C06042=1129.909,261.434,-70.854,-178.404,10.030,149.564
C06043=1129.914,261.185,-70.825,-178.407,10.028,149.564
C06044=1129.917,260.938,-70.797,-178.411,10.024,149.564
C06045=1129.922,260.689,-70.768,-178.414,10.021,149.564
C06046=1129.926,260.440,-70.738,-178.418,10.018,149.564
C06047=1129.931,260.192,-70.711,-178.421,10.015,149.565
C06048=1129.935,259.944,-70.681,-178.424,10.012,149.565
C06049=1129.939,259.695,-70.652,-178.428,10.010,149.565
C06050=1129.943,259.448,-70.624,-178.431,10.006,149.565
C06051=1129.948,259.199,-70.595,-178.434,10.003,149.565
C06052=1129.952,258.951,-70.566,-178.438,10.000,149.565
C06053=1129.956,258.702,-70.538,-178.441,9.997,149.565
C06054=1129.961,258.454,-70.509,-178.444,9.994,149.565
C06055=1129.965,258.206,-70.480,-178.447,9.991,149.566
C06056=1129.969,257.957,-70.452,-178.450,9.988,149.566
C06057=1129.974,257.709,-70.423,-178.453,9.985,149.566
C06058=1129.977,257.461,-70.394,-178.456,9.982,149.566
C06059=1129.982,257.212,-70.366,-178.459,9.980,149.566
C06060=1129.987,256.964,-70.337,-178.463,9.976,149.566
C06061=1129.990,256.716,-70.308,-178.465,9.973,149.566
C06062=1129.995,256.468,-70.280,-178.468,9.971,149.566
C06063=1129.999,256.219,-70.252,-178.471,9.968,149.566
C06064=1130.004,255.970,-70.223,-178.474,9.965,149.566
C06065=1130.008,255.723,-70.195,-178.473,9.964,149.566
C06066=1130.012,255.474,-70.166,-178.473,9.964,149.566
C06067=1130.016,255.226,-70.138,-178.472,9.963,149.565
C06068=1130.021,254.978,-70.109,-178.472,9.962,149.565
C06069=1130.024,254.730,-70.081,-178.472,9.961,149.565
C06070=1130.029,254.481,-70.052,-178.472,9.960,149.565
C06071=1130.033,254.233,-70.024,-178.473,9.959,149.565
C06072=1130.037,254.019,-70.000,-178.473,9.958,149.564
C06073=1130.041,253.805,-69.975,-178.475,9.956,149.564
C06074=1130.044,253.591,-69.950,-178.475,9.955,149.564
C06075=1130.048,253.377,-69.925,-178.476,9.954,149.564
C06076=1130.052,253.163,-69.901,-178.479,9.952,149.564
C06077=1130.055,252.950,-69.877,-178.480,9.950,149.564
C06078=1130.059,252.735,-69.853,-178.482,9.949,149.565
C06079=1130.063,252.522,-69.827,-178.484,9.947,149.565
C06080=1130.068,252.274,-69.799,-178.487,9.944,149.565
C06081=1130.072,252.025,-69.771,-178.489,9.942,149.565
C06082=1130.075,251.777,-69.743,-178.493,9.939,149.565
C06083=1130.080,251.529,-69.714,-178.496,9.936,149.565
C06084=1130.084,251.280,-69.686,-178.500,9.934,149.566
C06085=1130.089,251.032,-69.658,-178.504,9.931,149.566
C06086=1130.093,250.783,-69.630,-178.508,9.927,149.566
C06087=1130.098,250.535,-69.601,-178.512,9.924,149.567
C06088=1130.102,250.287,-69.573,-178.517,9.920,149.567
C06089=1130.106,250.039,-69.545,-178.522,9.916,149.567
C06090=1130.110,249.790,-69.516,-178.527,9.913,149.568
C06091=1130.115,249.541,-69.489,-178.533,9.908,149.568
C06092=1130.119,249.293,-69.461,-178.538,9.904,149.569
C06093=1130.123,249.044,-69.432,-178.544,9.900,149.569
C06094=1130.128,248.796,-69.404,-178.551,9.895,149.570
C06095=1130.131,248.548,-69.376,-178.557,9.890,149.570
C06096=1130.137,248.300,-69.348,-178.564,9.885,149.571
C06097=1130.141,248.052,-69.320,-178.570,9.880,149.571
C06098=1130.145,247.803,-69.293,-178.577,9.874,149.572
C06099=1130.149,247.555,-69.265,-178.585,9.869,149.572
C06100=1130.154,247.306,-69.236,-178.589,9.865,149.573
C06101=1130.158,247.058,-69.208,-178.590,9.863,149.573
C06102=1130.163,246.809,-69.181,-178.592,9.860,149.572
C06103=1130.167,246.561,-69.153,-178.593,9.858,149.572
C06104=1130.171,246.313,-69.125,-178.594,9.856,149.572
C06105=1130.176,246.063,-69.097,-178.595,9.854,149.572
C06106=1130.180,245.816,-69.069,-178.597,9.852,149.572
C06107=1130.184,245.568,-69.042,-178.598,9.850,149.571
C06108=1130.188,245.319,-69.014,-178.599,9.848,149.571
C06109=1130.193,245.071,-68.987,-178.601,9.845,149.571
C06110=1130.197,244.822,-68.958,-178.602,9.844,149.571
C06111=1130.201,244.574,-68.931,-178.604,9.841,149.571
C06112=1130.206,244.325,-68.903,-178.606,9.839,149.571
C06113=1130.210,244.076,-68.876,-178.607,9.837,149.571
C06114=1130.215,243.828,-68.848,-178.609,9.835,149.571
C06115=1130.219,243.580,-68.820,-178.610,9.833,149.571
C06116=1130.223,243.331,-68.793,-178.612,9.830,149.571
C06117=1130.227,243.083,-68.765,-178.614,9.829,149.571
C06118=1130.231,242.834,-68.737,-178.615,9.826,149.570
C06119=1130.236,242.586,-68.710,-178.617,9.824,149.570
C06120=1130.241,242.338,-68.682,-178.619,9.822,149.570
C06121=1130.244,242.089,-68.654,-178.621,9.819,149.570
C06122=1130.250,241.840,-68.627,-178.623,9.817,149.570
C06123=1130.254,241.593,-68.599,-178.625,9.815,149.570
C06124=1130.258,241.343,-68.571,-178.627,9.813,149.570
C06125=1130.262,241.096,-68.544,-178.629,9.810,149.570
C06126=1130.267,240.847,-68.517,-178.632,9.808,149.570
C06127=1130.271,240.598,-68.489,-178.634,9.805,149.570
C06128=1130.275,240.385,-68.466,-178.636,9.804,149.570
C06129=1130.279,240.171,-68.441,-178.638,9.802,149.570
C06130=1130.282,239.956,-68.418,-178.639,9.799,149.570
C06131=1130.286,239.743,-68.395,-178.642,9.797,149.571
C06132=1130.290,239.529,-68.371,-178.644,9.795,149.570
C06133=1130.293,239.315,-68.347,-178.646,9.793,149.571
C06134=1130.297,239.100,-68.323,-178.648,9.791,149.571
C06135=1130.301,238.887,-68.300,-178.650,9.789,149.571
C06136=1130.305,238.638,-68.272,-178.652,9.787,149.571
C06137=1130.310,238.390,-68.245,-178.655,9.784,149.571
C06138=1130.314,238.142,-68.217,-178.657,9.782,149.571
C06139=1130.319,237.893,-68.190,-178.660,9.779,149.571
C06140=1130.323,237.645,-68.162,-178.663,9.776,149.571
C06141=1130.327,237.396,-68.135,-178.665,9.774,149.571
C06142=1130.332,237.148,-68.108,-178.668,9.771,149.571
C06143=1130.336,236.900,-68.080,-178.671,9.768,149.571
C06144=1130.340,236.651,-68.053,-178.674,9.766,149.571
C06145=1130.344,236.402,-68.026,-178.677,9.763,149.572
C06146=1130.349,236.154,-67.999,-178.679,9.761,149.572
C06147=1130.353,235.906,-67.972,-178.682,9.758,149.572
C06148=1130.357,235.657,-67.944,-178.685,9.755,149.572
C06149=1130.362,235.408,-67.917,-178.688,9.752,149.572
C06150=1130.367,235.160,-67.890,-178.691,9.749,149.572
C06151=1130.371,234.911,-67.863,-178.694,9.746,149.572
C06152=1130.376,234.663,-67.835,-178.697,9.743,149.572
C06153=1130.379,234.415,-67.808,-178.700,9.741,149.572
C06154=1130.384,234.166,-67.781,-178.703,9.738,149.573
C06155=1130.388,233.918,-67.754,-178.707,9.735,149.573
C06156=1130.393,233.669,-67.727,-178.710,9.732,149.573
C06157=1130.398,233.421,-67.700,-178.713,9.729,149.573
C06158=1130.401,233.172,-67.673,-178.717,9.726,149.573
C06159=1130.406,232.923,-67.646,-178.719,9.723,149.573
C06160=1130.410,232.675,-67.619,-178.723,9.719,149.573
C06161=1130.415,232.426,-67.592,-178.726,9.717,149.574
C06162=1130.419,232.178,-67.566,-178.730,9.714,149.574
C06163=1130.423,231.930,-67.539,-178.734,9.710,149.574
C06164=1130.428,231.681,-67.512,-178.737,9.707,149.574
C06165=1130.433,231.433,-67.484,-178.740,9.704,149.574
C06166=1130.436,231.184,-67.458,-178.744,9.701,149.575
C06167=1130.441,230.935,-67.431,-178.748,9.697,149.575
C06168=1130.445,230.687,-67.404,-178.751,9.694,149.575
C06169=1130.449,230.438,-67.377,-178.754,9.691,149.575
C06170=1130.454,230.190,-67.350,-178.759,9.687,149.575
C06171=1130.459,229.941,-67.323,-178.762,9.683,149.575
C06172=1130.463,229.693,-67.296,-178.766,9.680,149.575
C06173=1130.467,229.445,-67.269,-178.770,9.677,149.576
C06174=1130.472,229.196,-67.243,-178.774,9.673,149.576
C06175=1130.476,228.947,-67.217,-178.777,9.670,149.576
C06176=1130.481,228.699,-67.190,-178.781,9.666,149.576
C06177=1130.485,228.451,-67.163,-178.784,9.663,149.576
C06178=1130.490,228.202,-67.137,-178.788,9.659,149.576
C06179=1130.494,227.954,-67.110,-178.792,9.656,149.576
C06180=1130.498,227.705,-67.083,-178.795,9.652,149.577
C06181=1130.503,227.457,-67.056,-178.799,9.648,149.577
C06182=1130.507,227.208,-67.030,-178.802,9.645,149.577
C06183=1130.512,226.959,-67.003,-178.806,9.641,149.577
C06184=1130.515,226.745,-66.980,-178.809,9.639,149.577
C06185=1130.520,226.531,-66.958,-178.811,9.636,149.577
C06186=1130.522,226.317,-66.936,-178.814,9.633,149.577
C06187=1130.526,226.103,-66.913,-178.817,9.630,149.577
C06188=1130.530,225.889,-66.890,-178.820,9.627,149.577
C06189=1130.534,225.675,-66.867,-178.823,9.623,149.577
C06190=1130.537,225.460,-66.844,-178.826,9.620,149.577
C06191=1130.542,225.246,-66.822,-178.829,9.618,149.577
C06192=1130.546,224.998,-66.794,-178.831,9.615,149.577
C06193=1130.550,224.749,-66.769,-178.835,9.611,149.577
C06194=1130.554,224.501,-66.742,-178.837,9.608,149.577
C06195=1130.559,224.252,-66.716,-178.841,9.604,149.578
C06196=1130.563,224.003,-66.689,-178.844,9.601,149.577
C06197=1130.568,223.754,-66.663,-178.847,9.598,149.578
C06198=1130.573,223.507,-66.637,-178.850,9.595,149.577
C06199=1130.577,223.258,-66.611,-178.853,9.591,149.577
C06200=1130.582,223.009,-66.585,-178.856,9.588,149.578
C06201=1130.586,222.761,-66.558,-178.859,9.584,149.577
C06202=1130.590,222.512,-66.533,-178.861,9.581,149.577
C06203=1130.595,222.263,-66.506,-178.864,9.578,149.577
C06204=1130.599,222.015,-66.480,-178.867,9.574,149.577
C06205=1130.603,221.766,-66.454,-178.870,9.571,149.577
C06206=1130.609,221.517,-66.428,-178.873,9.568,149.577
C06207=1130.613,221.269,-66.402,-178.875,9.565,149.577
C06208=1130.617,221.020,-66.376,-178.878,9.562,149.577
C06209=1130.622,220.771,-66.350,-178.880,9.559,149.577
C06210=1130.626,220.523,-66.323,-178.883,9.555,149.577
C06211=1130.630,220.274,-66.297,-178.886,9.552,149.577
C06212=1130.635,220.026,-66.272,-178.888,9.549,149.577
C06213=1130.640,219.777,-66.246,-178.891,9.545,149.577
C06214=1130.644,219.529,-66.219,-178.893,9.542,149.577
C06215=1130.648,219.280,-66.193,-178.895,9.540,149.577
C06216=1130.652,219.031,-66.168,-178.897,9.537,149.577
C06217=1130.657,218.783,-66.142,-178.900,9.534,149.576
C06218=1130.662,218.534,-66.116,-178.903,9.531,149.576
C06219=1130.666,218.286,-66.089,-178.905,9.527,149.576
C06220=1130.670,218.037,-66.064,-178.907,9.524,149.576
C06221=1130.674,217.788,-66.038,-178.909,9.522,149.576
C06222=1130.679,217.540,-66.013,-178.912,9.519,149.576
C06223=1130.683,217.291,-65.987,-178.914,9.515,149.576
C06224=1130.688,217.043,-65.961,-178.916,9.513,149.576
C06225=1130.692,216.793,-65.935,-178.918,9.510,149.576
C06226=1130.697,216.545,-65.909,-178.920,9.507,149.575
C06227=1130.702,216.297,-65.884,-178.922,9.504,149.575
C06228=1130.706,216.048,-65.858,-178.924,9.501,149.575
C06229=1130.710,215.799,-65.832,-178.926,9.498,149.575
C06230=1130.715,215.551,-65.807,-178.928,9.496,149.575
C06231=1130.719,215.302,-65.781,-178.930,9.492,149.575
C06232=1130.723,215.053,-65.755,-178.932,9.490,149.575
C06233=1130.727,214.804,-65.729,-178.934,9.487,149.574
C06234=1130.732,214.556,-65.704,-178.936,9.484,149.574
C06235=1130.737,214.307,-65.678,-178.938,9.481,149.574
C06236=1130.741,214.058,-65.652,-178.939,9.479,149.574
C06237=1130.746,213.810,-65.627,-178.941,9.476,149.574
C06238=1130.751,213.562,-65.601,-178.943,9.474,149.574
C06239=1130.755,213.313,-65.575,-178.945,9.471,149.574
C06240=1130.758,213.099,-65.554,-178.946,9.469,149.573
C06241=1130.762,212.885,-65.531,-178.947,9.467,149.573
C06242=1130.766,212.670,-65.508,-178.948,9.464,149.573
C06243=1130.770,212.456,-65.487,-178.950,9.463,149.573
C06244=1130.774,212.242,-65.465,-178.951,9.460,149.573
C06245=1130.778,212.028,-65.443,-178.952,9.459,149.573
C06246=1130.781,211.813,-65.421,-178.954,9.456,149.572
C06247=1130.785,211.600,-65.399,-178.956,9.454,149.572
C06248=1130.790,211.351,-65.374,-178.958,9.451,149.572
C06249=1130.794,211.102,-65.348,-178.960,9.449,149.572
C06250=1130.798,210.853,-65.323,-178.961,9.446,149.572
C06251=1130.803,210.605,-65.297,-178.963,9.444,149.572
C06252=1130.807,210.356,-65.271,-178.965,9.441,149.572
C06253=1130.812,210.108,-65.246,-178.967,9.439,149.572
C06254=1130.817,209.859,-65.221,-178.969,9.436,149.572
C06255=1130.821,209.610,-65.195,-178.971,9.434,149.572
C06256=1130.825,209.361,-65.170,-178.973,9.431,149.572
C06257=1130.830,209.113,-65.144,-178.976,9.428,149.572
C06258=1130.835,208.864,-65.119,-178.977,9.426,149.572
C06259=1130.839,208.616,-65.094,-178.979,9.424,149.572
C06260=1130.844,208.367,-65.068,-178.982,9.421,149.572
C06261=1130.848,208.118,-65.042,-178.984,9.419,149.572
C06262=1130.853,207.869,-65.018,-178.987,9.415,149.572
C06263=1130.856,207.621,-64.992,-178.990,9.413,149.572
C06264=1130.861,207.373,-64.967,-178.992,9.410,149.572
C06265=1130.866,207.123,-64.942,-178.995,9.408,149.572
C06266=1130.870,206.874,-64.916,-178.997,9.405,149.572
C06267=1130.875,206.626,-64.891,-178.999,9.403,149.572
C06268=1130.879,206.377,-64.866,-179.002,9.399,149.572
C06269=1130.884,206.129,-64.840,-179.005,9.397,149.572
C06270=1130.888,205.880,-64.815,-179.007,9.394,149.572
C06271=1130.893,205.632,-64.791,-179.010,9.391,149.572
C06272=1130.897,205.383,-64.765,-179.013,9.388,149.572
C06273=1130.902,205.133,-64.740,-179.016,9.385,149.572
C06274=1130.906,204.885,-64.714,-179.019,9.382,149.573
C06275=1130.911,204.636,-64.689,-179.022,9.380,149.573
C06276=1130.915,204.388,-64.665,-179.025,9.377,149.573
C06277=1130.920,204.139,-64.640,-179.027,9.374,149.573
C06278=1130.924,203.891,-64.614,-179.030,9.371,149.573
C06279=1130.929,203.641,-64.589,-179.034,9.367,149.573
C06280=1130.933,203.393,-64.564,-179.037,9.365,149.573
C06281=1130.938,203.144,-64.539,-179.040,9.362,149.573
C06282=1130.942,202.896,-64.514,-179.043,9.358,149.573
C06283=1130.946,202.647,-64.489,-179.046,9.356,149.574
C06284=1130.951,202.399,-64.464,-179.050,9.352,149.574
C06285=1130.956,202.149,-64.439,-179.053,9.349,149.574
C06286=1130.961,201.900,-64.414,-179.056,9.346,149.574
C06287=1130.964,201.652,-64.389,-179.060,9.342,149.574
C06288=1130.969,201.403,-64.365,-179.063,9.340,149.574
C06289=1130.974,201.155,-64.340,-179.066,9.336,149.574
C06290=1130.978,200.906,-64.315,-179.070,9.333,149.575
C06291=1130.983,200.657,-64.290,-179.074,9.329,149.575
C06292=1130.987,200.408,-64.266,-179.077,9.326,149.575
C06293=1130.992,200.160,-64.240,-179.080,9.323,149.575
C06294=1130.995,199.911,-64.216,-179.084,9.319,149.575
C06295=1131.001,199.662,-64.191,-179.088,9.316,149.576
C06296=1131.004,199.448,-64.170,-179.091,9.313,149.576
C06297=1131.008,199.234,-64.149,-179.094,9.310,149.576
C06298=1131.012,199.019,-64.127,-179.097,9.306,149.576
C06299=1131.016,198.805,-64.106,-179.100,9.303,149.576
C06300=1131.020,198.591,-64.085,-179.104,9.300,149.576
C06301=1131.024,198.376,-64.064,-179.107,9.297,149.576
C06302=1131.028,198.162,-64.042,-179.111,9.294,149.576
C06303=1131.032,197.947,-64.021,-179.113,9.291,149.577
C06304=1131.037,197.699,-63.997,-179.118,9.287,149.577
C06305=1131.040,197.450,-63.972,-179.122,9.283,149.577
C06306=1131.045,197.201,-63.948,-179.126,9.279,149.577
C06307=1131.050,196.953,-63.924,-179.130,9.275,149.577
C06308=1131.054,196.703,-63.899,-179.134,9.271,149.577
C06309=1131.059,196.455,-63.875,-179.138,9.267,149.578
C06310=1131.064,196.206,-63.850,-179.142,9.264,149.578
C06311=1131.068,195.957,-63.825,-179.143,9.261,149.577
C06312=1131.072,195.709,-63.801,-179.144,9.258,149.577
C06313=1131.077,195.460,-63.777,-179.146,9.257,149.577
C06314=1131.081,195.211,-63.752,-179.147,9.254,149.577
C06315=1131.086,194.962,-63.728,-179.149,9.251,149.577
C06316=1131.091,194.714,-63.704,-179.151,9.249,149.577
C06317=1131.095,194.465,-63.679,-179.152,9.246,149.576
C06318=1131.099,194.216,-63.654,-179.153,9.243,149.576
C06319=1131.104,193.967,-63.630,-179.155,9.241,149.576
C06320=1131.108,193.719,-63.606,-179.157,9.238,149.576
C06321=1131.113,193.470,-63.582,-179.159,9.236,149.576
C06322=1131.118,193.221,-63.558,-179.160,9.233,149.576
C06323=1131.122,192.972,-63.534,-179.162,9.231,149.576
C06324=1131.127,192.723,-63.509,-179.164,9.228,149.575
C06325=1131.131,192.475,-63.485,-179.165,9.226,149.575
C06326=1131.135,192.226,-63.461,-179.167,9.224,149.575
C06327=1131.140,191.977,-63.436,-179.169,9.221,149.575
C06328=1131.145,191.728,-63.413,-179.171,9.218,149.575
C06329=1131.149,191.480,-63.389,-179.173,9.216,149.575
C06330=1131.154,191.230,-63.364,-179.175,9.213,149.575
C06331=1131.158,190.982,-63.339,-179.177,9.211,149.575
C06332=1131.163,190.733,-63.315,-179.179,9.207,149.575
C06333=1131.167,190.484,-63.292,-179.181,9.205,149.575
C06334=1131.173,190.236,-63.267,-179.183,9.203,149.575
C06335=1131.176,189.987,-63.243,-179.185,9.199,149.574
C06336=1131.181,189.738,-63.220,-179.187,9.197,149.574
C06337=1131.186,189.489,-63.195,-179.189,9.194,149.574
C06338=1131.191,189.240,-63.171,-179.191,9.191,149.574
C06339=1131.195,188.992,-63.147,-179.194,9.188,149.574
C06340=1131.200,188.743,-63.123,-179.196,9.186,149.574
C06341=1131.204,188.494,-63.099,-179.198,9.183,149.574
C06342=1131.209,188.245,-63.074,-179.200,9.181,149.574
C06343=1131.213,187.996,-63.051,-179.203,9.178,149.574
C06344=1131.218,187.748,-63.027,-179.205,9.174,149.574
C06345=1131.222,187.499,-63.003,-179.207,9.172,149.574
C06346=1131.227,187.250,-62.979,-179.210,9.169,149.574
C06347=1131.232,187.002,-62.955,-179.212,9.166,149.574
C06348=1131.236,186.752,-62.931,-179.215,9.163,149.574
C06349=1131.240,186.503,-62.907,-179.218,9.160,149.574
C06350=1131.245,186.254,-62.884,-179.220,9.158,149.574
C06351=1131.250,186.006,-62.859,-179.222,9.155,149.574
C06352=1131.253,185.791,-62.839,-179.225,9.151,149.574
C06353=1131.257,185.577,-62.818,-179.227,9.149,149.574
C06354=1131.262,185.363,-62.798,-179.228,9.147,149.574
C06355=1131.265,185.149,-62.777,-179.231,9.144,149.574
C06356=1131.269,184.934,-62.757,-179.233,9.142,149.574
C06357=1131.273,184.719,-62.737,-179.236,9.139,149.574
C06358=1131.277,184.504,-62.716,-179.238,9.136,149.574
C06359=1131.282,184.290,-62.695,-179.240,9.133,149.574
C06360=1131.286,184.042,-62.671,-179.243,9.130,149.574
C06361=1131.290,183.792,-62.648,-179.246,9.127,149.574
C06362=1131.295,183.543,-62.624,-179.248,9.124,149.574
C06363=1131.299,183.295,-62.600,-179.251,9.122,149.574
C06364=1131.304,183.046,-62.577,-179.254,9.118,149.574
C06365=1131.308,182.797,-62.553,-179.257,9.115,149.574
C06366=1131.313,182.548,-62.529,-179.259,9.111,149.574
C06367=1131.318,182.299,-62.506,-179.263,9.108,149.574
C06368=1131.322,182.051,-62.482,-179.265,9.105,149.574
C06369=1131.327,181.802,-62.459,-179.268,9.102,149.574
C06370=1131.332,181.553,-62.435,-179.272,9.098,149.574
C06371=1131.336,181.304,-62.411,-179.274,9.095,149.574
C06372=1131.341,181.055,-62.388,-179.278,9.092,149.574
C06373=1131.345,180.807,-62.365,-179.280,9.088,149.574
C06374=1131.349,180.558,-62.342,-179.283,9.085,149.574
C06375=1131.354,180.309,-62.318,-179.287,9.081,149.574
C06376=1131.358,180.060,-62.294,-179.290,9.078,149.574
C06377=1131.363,179.811,-62.271,-179.293,9.074,149.574
C06378=1131.368,179.562,-62.248,-179.296,9.071,149.574
C06379=1131.372,179.313,-62.224,-179.299,9.067,149.574
C06380=1131.377,179.064,-62.201,-179.302,9.064,149.574
C06381=1131.382,178.816,-62.177,-179.304,9.061,149.574
C06382=1131.386,178.567,-62.154,-179.306,9.058,149.574
C06383=1131.390,178.318,-62.131,-179.308,9.055,149.574
C06384=1131.396,178.069,-62.108,-179.310,9.052,149.574
C06385=1131.400,177.820,-62.084,-179.313,9.049,149.574
C06386=1131.405,177.571,-62.061,-179.314,9.047,149.574
C06387=1131.409,177.323,-62.038,-179.317,9.043,149.574
C06388=1131.414,177.074,-62.015,-179.319,9.041,149.574
C06389=1131.418,176.825,-61.991,-179.321,9.038,149.573
C06390=1131.423,176.576,-61.968,-179.323,9.034,149.573
C06391=1131.428,176.327,-61.945,-179.325,9.032,149.573
C06392=1131.432,176.078,-61.922,-179.327,9.029,149.573
C06393=1131.436,175.829,-61.899,-179.330,9.026,149.573
C06394=1131.441,175.580,-61.875,-179.332,9.023,149.573
C06395=1131.446,175.331,-61.852,-179.334,9.020,149.573
C06396=1131.450,175.083,-61.829,-179.336,9.017,149.573
C06397=1131.455,174.834,-61.806,-179.338,9.014,149.573
C06398=1131.460,174.585,-61.783,-179.340,9.011,149.572
C06399=1131.464,174.336,-61.759,-179.343,9.008,149.572
C06400=1131.468,174.087,-61.737,-179.345,9.005,149.572
C06401=1131.473,173.838,-61.713,-179.347,9.002,149.572
C06402=1131.478,173.590,-61.690,-179.349,8.999,149.572
C06403=1131.482,173.341,-61.668,-179.352,8.996,149.572
C06404=1131.487,173.091,-61.645,-179.354,8.993,149.572
C06405=1131.492,172.842,-61.622,-179.356,8.990,149.572
C06406=1131.496,172.593,-61.599,-179.358,8.987,149.572
C06407=1131.501,172.344,-61.575,-179.361,8.984,149.572
C06408=1131.505,172.130,-61.556,-179.363,8.981,149.572
C06409=1131.509,171.916,-61.536,-179.365,8.979,149.572
C06410=1131.513,171.701,-61.516,-179.367,8.976,149.571
C06411=1131.517,171.486,-61.496,-179.369,8.973,149.571
C06412=1131.521,171.272,-61.477,-179.371,8.971,149.571
C06413=1131.525,171.057,-61.457,-179.373,8.969,149.571
C06414=1131.528,170.843,-61.437,-179.375,8.965,149.571
C06415=1131.533,170.628,-61.418,-179.377,8.963,149.571
C06416=1131.537,170.379,-61.395,-179.379,8.960,149.571
C06417=1131.542,170.130,-61.371,-179.382,8.957,149.571
C06418=1131.547,169.882,-61.350,-179.384,8.953,149.571
C06419=1131.552,169.633,-61.326,-179.386,8.951,149.571
C06420=1131.556,169.384,-61.303,-179.388,8.948,149.571
C06421=1131.561,169.134,-61.281,-179.391,8.945,149.571
C06422=1131.565,168.886,-61.258,-179.393,8.941,149.571
C06423=1131.570,168.637,-61.235,-179.395,8.938,149.570
C06424=1131.574,168.388,-61.213,-179.398,8.935,149.570
C06425=1131.579,168.139,-61.190,-179.400,8.932,149.570
C06426=1131.584,167.890,-61.168,-179.403,8.929,149.570
C06427=1131.588,167.641,-61.145,-179.405,8.925,149.570
C06428=1131.592,167.392,-61.122,-179.407,8.922,149.570
C06429=1131.598,167.143,-61.100,-179.410,8.919,149.570
C06430=1131.602,166.895,-61.077,-179.412,8.916,149.570
C06431=1131.607,166.645,-61.054,-179.415,8.913,149.570
C06432=1131.611,166.396,-61.031,-179.417,8.909,149.570
C06433=1131.616,166.147,-61.009,-179.420,8.906,149.570
C06434=1131.620,165.899,-60.986,-179.422,8.903,149.570
C06435=1131.625,165.649,-60.964,-179.425,8.900,149.570
C06436=1131.630,165.401,-60.941,-179.427,8.897,149.570
C06437=1131.635,165.151,-60.919,-179.429,8.893,149.569
C06438=1131.639,164.903,-60.896,-179.432,8.890,149.569
C06439=1131.644,164.654,-60.874,-179.434,8.887,149.569
C06440=1131.648,164.405,-60.851,-179.437,8.884,149.569
C06441=1131.653,164.156,-60.829,-179.439,8.880,149.569
C06442=1131.658,163.907,-60.807,-179.441,8.877,149.569
C06443=1131.662,163.658,-60.784,-179.444,8.874,149.569
C06444=1131.667,163.409,-60.762,-179.446,8.871,149.569
C06445=1131.671,163.161,-60.739,-179.449,8.868,149.569
C06446=1131.676,162.911,-60.717,-179.451,8.865,149.569
C06447=1131.681,162.662,-60.695,-179.454,8.861,149.569
C06448=1131.685,162.414,-60.672,-179.457,8.858,149.569
C06449=1131.691,162.165,-60.650,-179.459,8.854,149.569
C06450=1131.695,161.915,-60.628,-179.461,8.851,149.568
C06451=1131.699,161.667,-60.605,-179.464,8.848,149.568
C06452=1131.704,161.418,-60.583,-179.466,8.845,149.568
C06453=1131.709,161.168,-60.561,-179.470,8.841,149.568
C06454=1131.714,160.920,-60.539,-179.472,8.837,149.568
C06455=1131.718,160.671,-60.516,-179.474,8.834,149.568
C06456=1131.723,160.421,-60.494,-179.477,8.831,149.568
C06457=1131.727,160.173,-60.472,-179.479,8.828,149.568
C06458=1131.732,159.923,-60.450,-179.482,8.824,149.568
C06459=1131.737,159.675,-60.428,-179.484,8.821,149.568
C06460=1131.741,159.426,-60.406,-179.487,8.818,149.568
C06461=1131.746,159.177,-60.383,-179.490,8.813,149.567
C06462=1131.750,158.928,-60.361,-179.492,8.810,149.567
C06463=1131.755,158.679,-60.340,-179.495,8.807,149.567
C06464=1131.759,158.464,-60.320,-179.497,8.804,149.567
C06465=1131.763,158.249,-60.302,-179.499,8.801,149.567
C06466=1131.767,158.035,-60.283,-179.501,8.798,149.567
C06467=1131.771,157.820,-60.263,-179.504,8.795,149.567
C06468=1131.775,157.605,-60.245,-179.506,8.792,149.567
C06469=1131.779,157.391,-60.226,-179.508,8.789,149.567
C06470=1131.783,157.176,-60.207,-179.510,8.786,149.567
C06471=1131.787,156.961,-60.188,-179.513,8.783,149.567
C06472=1131.792,156.713,-60.166,-179.515,8.780,149.567
C06473=1131.796,156.464,-60.144,-179.518,8.776,149.566
C06474=1131.801,156.215,-60.123,-179.521,8.773,149.566
C06475=1131.806,155.965,-60.100,-179.523,8.768,149.566
C06476=1131.811,155.717,-60.078,-179.526,8.765,149.566
C06477=1131.815,155.467,-60.056,-179.529,8.761,149.566
C06478=1131.820,155.219,-60.034,-179.531,8.758,149.566
C06479=1131.824,154.969,-60.012,-179.534,8.755,149.566
C06480=1131.829,154.721,-59.991,-179.537,8.751,149.566
C06481=1131.834,154.471,-59.970,-179.539,8.747,149.566
C06482=1131.839,154.222,-59.948,-179.542,8.743,149.566
C06483=1131.844,153.973,-59.926,-179.544,8.740,149.566
C06484=1131.848,153.724,-59.904,-179.547,8.736,149.565
C06485=1131.853,153.475,-59.882,-179.550,8.732,149.565
C06486=1131.858,153.227,-59.861,-179.552,8.729,149.565
C06487=1131.862,152.977,-59.839,-179.556,8.725,149.565
C06488=1131.867,152.728,-59.818,-179.558,8.722,149.565
C06489=1131.872,152.480,-59.796,-179.561,8.717,149.565
C06490=1131.876,152.230,-59.774,-179.563,8.714,149.565
C06491=1131.881,151.981,-59.753,-179.566,8.710,149.565
C06492=1131.886,151.732,-59.731,-179.569,8.706,149.564
C06493=1131.890,151.483,-59.710,-179.571,8.703,149.564
C06494=1131.895,151.235,-59.688,-179.574,8.699,149.564
C06495=1131.900,150.985,-59.667,-179.577,8.695,149.564
C06496=1131.904,150.736,-59.645,-179.580,8.691,149.564
C06497=1131.909,150.487,-59.623,-179.583,8.688,149.564
C06498=1131.914,150.238,-59.602,-179.586,8.683,149.564
C06499=1131.918,149.989,-59.580,-179.588,8.680,149.564
C06500=1131.923,149.739,-59.559,-179.591,8.676,149.563
C06501=1131.928,149.491,-59.538,-179.593,8.672,149.563
C06502=1131.932,149.243,-59.517,-179.596,8.669,149.563
C06503=1131.937,148.993,-59.495,-179.599,8.664,149.563
C06504=1131.942,148.744,-59.474,-179.602,8.660,149.563
C06505=1131.947,148.495,-59.453,-179.605,8.656,149.563
C06506=1131.951,148.246,-59.431,-179.608,8.652,149.563
C06507=1131.956,147.996,-59.410,-179.610,8.649,149.562
C06508=1131.961,147.748,-59.389,-179.613,8.645,149.562
C06509=1131.966,147.498,-59.368,-179.616,8.641,149.562
C06510=1131.970,147.250,-59.346,-179.618,8.636,149.562
C06511=1131.975,147.000,-59.325,-179.622,8.633,149.562
C06512=1131.979,146.752,-59.303,-179.624,8.628,149.562
C06513=1131.985,146.502,-59.283,-179.627,8.625,149.562
C06514=1131.989,146.253,-59.262,-179.629,8.621,149.561
C06515=1131.994,146.005,-59.240,-179.632,8.617,149.561
C06516=1131.998,145.755,-59.219,-179.635,8.613,149.561
C06517=1132.003,145.506,-59.199,-179.638,8.608,149.561
C06518=1132.008,145.257,-59.177,-179.641,8.604,149.561
C06519=1132.013,145.008,-59.156,-179.644,8.600,149.561
C06520=1132.017,144.793,-59.138,-179.645,8.597,149.560
C06521=1132.021,144.579,-59.120,-179.646,8.595,149.560
C06522=1132.025,144.364,-59.102,-179.647,8.591,149.560
C06523=1132.029,144.149,-59.084,-179.649,8.589,149.559
C06524=1132.033,143.934,-59.065,-179.649,8.586,149.559
C06525=1132.036,143.719,-59.047,-179.651,8.584,149.559
C06526=1132.041,143.504,-59.029,-179.652,8.581,149.558
C06527=1132.045,143.290,-59.011,-179.653,8.578,149.558
C06528=1132.050,143.041,-58.990,-179.655,8.574,149.558
C06529=1132.054,142.792,-58.970,-179.656,8.571,149.557
C06530=1132.059,142.542,-58.949,-179.657,8.568,149.557
C06531=1132.064,142.293,-58.928,-179.659,8.564,149.557
C06532=1132.069,142.045,-58.907,-179.660,8.562,149.556
C06533=1132.073,141.795,-58.885,-179.662,8.558,149.556
C06534=1132.078,141.546,-58.865,-179.663,8.555,149.555
C06535=1132.083,141.297,-58.844,-179.665,8.551,149.555
C06536=1132.087,141.048,-58.824,-179.666,8.548,149.555
C06537=1132.092,140.798,-58.803,-179.668,8.545,149.555
C06538=1132.097,140.550,-58.782,-179.669,8.542,149.554
C06539=1132.102,140.301,-58.761,-179.671,8.539,149.554
C06540=1132.106,140.052,-58.740,-179.672,8.535,149.553
C06541=1132.111,139.803,-58.719,-179.673,8.532,149.553
C06542=1132.116,139.554,-58.699,-179.675,8.528,149.553
C06543=1132.121,139.304,-58.678,-179.676,8.525,149.552
C06544=1132.125,139.055,-58.657,-179.678,8.523,149.552
C06545=1132.130,138.806,-58.636,-179.679,8.519,149.552
C06546=1132.134,138.557,-58.616,-179.681,8.516,149.552
C06547=1132.140,138.307,-58.595,-179.683,8.512,149.551
C06548=1132.144,138.058,-58.575,-179.684,8.509,149.551
C06549=1132.149,137.810,-58.553,-179.686,8.506,149.550
C06550=1132.153,137.561,-58.533,-179.687,8.503,149.550
C06551=1132.158,137.312,-58.512,-179.689,8.499,149.550
C06552=1132.163,137.063,-58.491,-179.690,8.496,149.550
C06553=1132.167,136.814,-58.471,-179.692,8.492,149.549
C06554=1132.173,136.564,-58.450,-179.693,8.490,149.549
C06555=1132.177,136.315,-58.430,-179.695,8.486,149.549
C06556=1132.182,136.066,-58.409,-179.696,8.483,149.548
C06557=1132.187,135.817,-58.389,-179.698,8.480,149.548
C06558=1132.191,135.568,-58.369,-179.699,8.476,149.548
C06559=1132.197,135.318,-58.348,-179.701,8.473,149.547
C06560=1132.201,135.069,-58.327,-179.702,8.470,149.547
C06561=1132.205,134.821,-58.307,-179.705,8.466,149.547
C06562=1132.211,134.571,-58.286,-179.706,8.464,149.546
C06563=1132.215,134.322,-58.265,-179.708,8.460,149.546
C06564=1132.219,134.073,-58.245,-179.709,8.457,149.546
C06565=1132.225,133.824,-58.224,-179.711,8.453,149.545
C06566=1132.229,133.575,-58.204,-179.712,8.451,149.545
C06567=1132.234,133.326,-58.184,-179.714,8.447,149.545
C06568=1132.239,133.076,-58.163,-179.716,8.443,149.545
C06569=1132.243,132.827,-58.143,-179.717,8.440,149.544
C06570=1132.248,132.578,-58.122,-179.719,8.437,149.544
C06571=1132.253,132.329,-58.101,-179.720,8.434,149.544
C06572=1132.258,132.080,-58.082,-179.722,8.430,149.543
C06573=1132.263,131.831,-58.062,-179.724,8.428,149.543
C06574=1132.268,131.582,-58.041,-179.726,8.424,149.543
C06575=1132.272,131.333,-58.020,-179.728,8.420,149.543
C06576=1132.279,130.949,-57.989,-179.730,8.416,149.542
C06577=1132.287,130.563,-57.958,-179.733,8.410,149.542
C06578=1132.294,130.179,-57.927,-179.735,8.406,149.541
C06579=1132.302,129.795,-57.895,-179.738,8.400,149.541
C06580=1132.322,128.765,-57.809,-179.030,7.005,149.019
C06581=1132.326,128.516,-57.789,-179.033,7.003,149.019
C06582=1132.331,128.266,-57.769,-179.036,7.001,149.019
C06583=1132.335,128.017,-57.749,-179.038,7.000,149.020
C06584=1132.341,127.768,-57.730,-179.042,6.997,149.020
C06585=1132.345,127.519,-57.710,-179.044,6.996,149.021
C06586=1132.350,127.270,-57.690,-179.047,6.993,149.021
C06587=1132.355,127.021,-57.670,-179.049,6.992,149.021
C06588=1132.360,126.771,-57.651,-179.052,6.990,149.022
C06589=1132.364,126.523,-57.631,-179.055,6.988,149.022
C06590=1132.368,126.273,-57.611,-179.058,6.986,149.022
C06591=1132.374,126.024,-57.592,-179.061,6.984,149.023
C06592=1132.379,125.775,-57.572,-179.064,6.983,149.023
C06593=1132.383,125.526,-57.552,-179.066,6.981,149.024
C06594=1132.388,125.277,-57.533,-179.069,6.979,149.024
C06595=1132.393,125.027,-57.513,-179.072,6.977,149.024
C06596=1132.398,124.778,-57.493,-179.075,6.975,149.025
C06597=1132.403,124.528,-57.474,-179.078,6.973,149.025
C06598=1132.408,124.280,-57.454,-179.081,6.972,149.026
C06599=1132.412,124.030,-57.434,-179.083,6.970,149.026
C06600=1132.416,123.781,-57.415,-179.086,6.968,149.026
C06601=1132.422,123.532,-57.396,-179.089,6.966,149.027
C06602=1132.426,123.283,-57.376,-179.092,6.964,149.027
C06603=1132.431,123.033,-57.356,-179.095,6.962,149.028
C06604=1132.436,122.785,-57.336,-179.098,6.961,149.028
C06605=1132.441,122.535,-57.317,-179.100,6.959,149.028
C06606=1132.446,122.287,-57.298,-179.103,6.957,149.029
C06607=1132.450,122.037,-57.278,-179.106,6.956,149.029
C06608=1132.455,121.788,-57.259,-179.109,6.953,149.030
C06609=1132.460,121.539,-57.239,-179.112,6.952,149.030
C06610=1132.465,121.289,-57.220,-179.115,6.950,149.030
C06611=1132.469,121.040,-57.201,-179.117,6.948,149.031
C06612=1132.474,120.791,-57.181,-179.120,6.946,149.031
C06613=1132.479,120.541,-57.162,-179.123,6.945,149.032
C06614=1132.485,120.293,-57.143,-179.125,6.943,149.032
C06615=1132.489,120.043,-57.123,-179.128,6.941,149.032
C06616=1132.494,119.794,-57.104,-179.132,6.939,149.033
C06617=1132.499,119.545,-57.085,-179.134,6.937,149.033
C06618=1132.503,119.295,-57.065,-179.137,6.936,149.034
C06619=1132.508,119.047,-57.046,-179.140,6.934,149.034
C06620=1132.513,118.797,-57.027,-179.142,6.932,149.034
C06621=1132.518,118.548,-57.007,-179.145,6.931,149.035
C06622=1132.523,118.299,-56.988,-179.148,6.929,149.035
C06623=1132.527,118.050,-56.969,-179.151,6.927,149.036
C06624=1132.532,117.801,-56.949,-179.153,6.926,149.036
C06625=1132.537,117.552,-56.930,-179.157,6.923,149.036
C06626=1132.542,117.302,-56.912,-179.159,6.921,149.037
C06627=1132.547,117.052,-56.892,-179.162,6.920,149.037
C06628=1132.552,116.803,-56.873,-179.165,6.918,149.038
C06629=1132.556,116.554,-56.854,-179.168,6.916,149.038
C06630=1132.561,116.305,-56.834,-179.170,6.915,149.038
C06631=1132.566,116.056,-56.815,-179.173,6.913,149.039
C06632=1132.571,115.807,-56.797,-179.176,6.911,149.039
C06633=1132.576,115.557,-56.777,-179.179,6.910,149.040
C06634=1132.580,115.308,-56.758,-179.181,6.908,149.040
C06635=1132.585,115.059,-56.739,-179.185,6.905,149.041
C06636=1132.590,114.810,-56.719,-179.187,6.904,149.041
C06637=1132.595,114.561,-56.701,-179.190,6.902,149.041
C06638=1132.600,114.311,-56.682,-179.193,6.900,149.042
C06639=1132.605,114.063,-56.663,-179.196,6.899,149.042
C06640=1132.610,113.812,-56.644,-179.198,6.897,149.043
C06641=1132.614,113.564,-56.625,-179.201,6.895,149.043
C06642=1132.619,113.314,-56.606,-179.204,6.894,149.043
C06643=1132.624,113.065,-56.586,-179.206,6.892,149.044
C06644=1132.629,112.816,-56.568,-179.209,6.890,149.044
C06645=1132.634,112.567,-56.549,-179.212,6.889,149.045
C06646=1132.638,112.317,-56.530,-179.215,6.887,149.045
C06647=1132.644,112.068,-56.511,-179.217,6.885,149.045
C06648=1132.648,111.819,-56.492,-179.220,6.884,149.046
C06649=1132.653,111.569,-56.474,-179.223,6.881,149.046
C06650=1132.658,111.321,-56.455,-179.226,6.880,149.047
C06651=1132.663,111.071,-56.435,-179.229,6.878,149.047
C06652=1132.668,110.822,-56.417,-179.232,6.876,149.047
C06653=1132.673,110.573,-56.398,-179.234,6.875,149.048
C06654=1132.677,110.323,-56.380,-179.237,6.873,149.048
C06655=1132.683,110.074,-56.360,-179.240,6.871,149.049
C06656=1132.687,109.825,-56.342,-179.243,6.869,149.049
C06657=1132.691,109.576,-56.323,-179.245,6.868,149.049
C06658=1132.697,109.326,-56.305,-179.249,6.867,149.050
C06659=1132.701,109.077,-56.286,-179.251,6.865,149.051
C06660=1132.707,108.828,-56.267,-179.254,6.863,149.051
C06661=1132.711,108.579,-56.248,-179.257,6.861,149.051
C06662=1132.716,108.329,-56.230,-179.259,6.860,149.052
C06663=1132.721,108.080,-56.211,-179.262,6.858,149.052
C06664=1132.726,107.831,-56.193,-179.265,6.856,149.053
C06665=1132.731,107.582,-56.173,-179.268,6.855,149.053
C06666=1132.736,107.332,-56.155,-179.270,6.853,149.053
C06667=1132.741,107.083,-56.137,-179.273,6.851,149.054
C06668=1132.745,106.834,-56.117,-179.276,6.850,149.054
C06669=1132.750,106.585,-56.099,-179.279,6.848,149.055
C06670=1132.755,106.336,-56.081,-179.281,6.846,149.055
C06671=1132.760,106.086,-56.062,-179.284,6.845,149.055
C06672=1132.765,105.837,-56.044,-179.287,6.843,149.056
C06673=1132.770,105.569,-56.024,-179.290,6.842,149.057
C06674=1132.775,105.300,-56.004,-179.293,6.839,149.057
C06675=1132.780,105.031,-55.984,-179.296,6.838,149.057
C06676=1132.786,104.763,-55.964,-179.299,6.836,149.058
C06677=1132.790,104.514,-55.945,-179.302,6.834,149.058
C06678=1132.795,104.265,-55.927,-179.304,6.833,149.059
C06679=1132.800,104.015,-55.908,-179.308,6.831,149.059
C06680=1132.805,103.766,-55.890,-179.310,6.830,149.060
C06681=1132.810,103.517,-55.872,-179.313,6.828,149.060
C06682=1132.815,103.268,-55.854,-179.316,6.826,149.060
C06683=1132.820,103.018,-55.835,-179.319,6.825,149.061
C06684=1132.825,102.769,-55.817,-179.321,6.823,149.061
C06685=1132.829,102.520,-55.798,-179.324,6.821,149.062
C06686=1132.834,102.271,-55.780,-179.327,6.820,149.062
C06687=1132.839,102.022,-55.762,-179.329,6.818,149.063
C06688=1132.844,101.772,-55.743,-179.332,6.816,149.063
C06689=1132.849,101.522,-55.725,-179.335,6.815,149.063
C06690=1132.854,101.274,-55.706,-179.338,6.813,149.064
C06691=1132.859,101.025,-55.688,-179.341,6.812,149.064
C06692=1132.863,100.775,-55.670,-179.344,6.810,149.065
C06693=1132.868,100.525,-55.652,-179.346,6.808,149.065
C06694=1132.873,100.276,-55.634,-179.349,6.807,149.066
C06695=1132.878,100.027,-55.616,-179.352,6.805,149.066
C06696=1132.883,99.778,-55.598,-179.355,6.803,149.066
C06697=1132.888,99.529,-55.580,-179.357,6.802,149.067
C06698=1132.892,99.279,-55.561,-179.360,6.800,149.067
C06699=1132.897,99.030,-55.543,-179.363,6.798,149.068
C06700=1132.902,98.780,-55.525,-179.366,6.797,149.068
C06701=1132.907,98.532,-55.507,-179.369,6.795,149.069
C06702=1132.913,98.282,-55.488,-179.372,6.794,149.069
C06703=1132.917,98.033,-55.470,-179.374,6.792,149.070
C06704=1132.922,97.783,-55.452,-179.376,6.791,149.070
C06705=1132.927,97.534,-55.434,-179.379,6.790,149.070
C06706=1132.932,97.285,-55.416,-179.382,6.788,149.071
C06707=1132.936,97.036,-55.398,-179.385,6.786,149.071
C06708=1132.942,96.786,-55.381,-179.387,6.785,149.072
C06709=1132.947,96.537,-55.363,-179.391,6.783,149.072
C06710=1132.952,96.288,-55.345,-179.393,6.782,149.073
C06711=1132.956,96.038,-55.327,-179.396,6.780,149.073
C06712=1132.961,95.789,-55.308,-179.399,6.778,149.074
C06713=1132.966,95.539,-55.290,-179.402,6.777,149.074
C06714=1132.971,95.290,-55.272,-179.404,6.775,149.074
C06715=1132.975,95.041,-55.254,-179.407,6.773,149.075
C06716=1132.980,94.792,-55.236,-179.410,6.772,149.075
C06717=1132.985,94.543,-55.218,-179.413,6.770,149.076
C06718=1132.991,94.293,-55.201,-179.416,6.769,149.076
C06719=1132.995,94.044,-55.183,-179.418,6.768,149.077
C06720=1133.000,93.795,-55.165,-179.421,6.766,149.077
C06721=1133.005,93.545,-55.147,-179.423,6.764,149.078
C06722=1133.010,93.296,-55.129,-179.426,6.763,149.078
C06723=1133.015,93.047,-55.111,-179.429,6.761,149.078
C06724=1133.020,92.797,-55.094,-179.432,6.759,149.079
C06725=1133.025,92.548,-55.076,-179.435,6.758,149.080
C06726=1133.030,92.299,-55.058,-179.438,6.757,149.080
C06727=1133.034,92.050,-55.041,-179.440,6.755,149.080
C06728=1133.039,91.800,-55.023,-179.443,6.753,149.081
C06729=1133.044,91.550,-55.005,-179.446,6.752,149.081
C06730=1133.049,91.301,-54.987,-179.448,6.751,149.082
C06731=1133.054,91.052,-54.969,-179.451,6.749,149.082
C06732=1133.059,90.802,-54.952,-179.454,6.748,149.083
C06733=1133.064,90.553,-54.934,-179.457,6.746,149.083
C06734=1133.069,90.304,-54.916,-179.459,6.744,149.084
C06735=1133.073,90.054,-54.899,-179.462,6.743,149.084
C06736=1133.078,89.805,-54.881,-179.465,6.741,149.084
C06737=1133.083,89.556,-54.863,-179.468,6.739,149.085
C06738=1133.088,89.306,-54.846,-179.470,6.738,149.085
C06739=1133.093,89.057,-54.828,-179.473,6.737,149.086
C06740=1133.099,88.808,-54.811,-179.476,6.736,149.086
C06741=1133.103,88.559,-54.794,-179.478,6.734,149.087
C06742=1133.108,88.310,-54.776,-179.481,6.732,149.087
C06743=1133.113,88.060,-54.758,-179.484,6.731,149.088
C06744=1133.118,87.811,-54.740,-179.487,6.729,149.088
C06745=1133.123,87.561,-54.724,-179.490,6.728,149.089
C06746=1133.128,87.312,-54.706,-179.493,6.726,149.089
C06747=1133.133,87.062,-54.688,-179.495,6.725,149.090
C06748=1133.138,86.813,-54.671,-179.498,6.724,149.090
C06749=1133.142,86.564,-54.653,-179.500,6.722,149.090
C06750=1133.147,86.315,-54.636,-179.503,6.720,149.091
C06751=1133.152,86.065,-54.618,-179.506,6.719,149.091
C06752=1133.157,85.816,-54.601,-179.509,6.717,149.092
C06753=1133.162,85.566,-54.584,-179.512,6.716,149.092
C06754=1133.167,85.317,-54.566,-179.514,6.715,149.093
C06755=1133.172,85.068,-54.549,-179.517,6.713,149.093
C06756=1133.177,84.819,-54.532,-179.519,6.711,149.094
C06757=1133.182,84.569,-54.514,-179.523,6.710,149.094
C06758=1133.187,84.320,-54.496,-179.525,6.708,149.095
C06759=1133.192,84.070,-54.479,-179.528,6.707,149.095
C06760=1133.196,83.821,-54.462,-179.530,6.706,149.095
C06761=1133.201,83.572,-54.445,-179.533,6.704,149.096
C06762=1133.206,83.322,-54.428,-179.536,6.703,149.096
C06763=1133.211,83.074,-54.410,-179.539,6.701,149.097
C06764=1133.217,82.824,-54.393,-179.542,6.700,149.097
C06765=1133.221,82.574,-54.376,-179.544,6.698,149.098
C06766=1133.226,82.325,-54.358,-179.547,6.697,149.098
C06767=1133.231,82.075,-54.341,-179.549,6.696,149.099
C06768=1133.236,81.826,-54.324,-179.552,6.694,149.099
C06769=1133.241,81.577,-54.307,-179.555,6.693,149.100
C06770=1133.246,81.328,-54.290,-179.558,6.691,149.100
C06771=1133.251,81.078,-54.273,-179.561,6.689,149.101
C06772=1133.256,80.829,-54.255,-179.563,6.688,149.101
C06773=1133.260,80.580,-54.238,-179.566,6.687,149.101
C06774=1133.265,80.330,-54.221,-179.569,6.686,149.102
C06775=1133.271,80.081,-54.205,-179.572,6.684,149.103
C06776=1133.275,79.832,-54.187,-179.574,6.682,149.103
C06777=1133.280,79.563,-54.169,-179.577,6.681,149.103
C06778=1133.286,79.295,-54.150,-179.580,6.679,149.104
C06779=1133.291,79.026,-54.132,-179.583,6.678,149.104
C06780=1133.296,78.758,-54.113,-179.586,6.676,149.105
C06781=1133.302,78.509,-54.097,-179.589,6.676,149.106
C06782=1133.306,78.259,-54.080,-179.591,6.674,149.106
C06783=1133.312,78.009,-54.063,-179.594,6.672,149.106
C06784=1133.316,77.760,-54.046,-179.597,6.671,149.107
C06785=1133.322,77.511,-54.028,-179.600,6.669,149.107
C06786=1133.326,77.262,-54.012,-179.602,6.668,149.108
C06787=1133.331,77.012,-53.994,-179.605,6.667,149.108
C06788=1133.336,76.763,-53.978,-179.608,6.665,149.109
C06789=1133.342,76.513,-53.961,-179.610,6.663,149.109
C06790=1133.346,76.264,-53.944,-179.613,6.662,149.110
C06791=1133.351,76.014,-53.927,-179.616,6.661,149.110
C06792=1133.356,75.765,-53.911,-179.619,6.660,149.111
C06793=1133.361,75.516,-53.894,-179.621,6.658,149.111
C06794=1133.366,75.266,-53.877,-179.624,6.656,149.112
C06795=1133.371,75.017,-53.860,-179.626,6.656,149.112
C06796=1133.376,74.768,-53.844,-179.629,6.654,149.113
C06797=1133.381,74.518,-53.826,-179.632,6.653,149.113
C06798=1133.385,74.269,-53.810,-179.635,6.651,149.114
C06799=1133.391,74.019,-53.793,-179.638,6.649,149.114
C06800=1133.396,73.770,-53.776,-179.640,6.649,149.115
C06801=1133.400,73.520,-53.760,-179.643,6.647,149.115
C06802=1133.406,73.271,-53.743,-179.646,6.646,149.116
C06803=1133.410,73.022,-53.726,-179.649,6.644,149.116
C06804=1133.415,72.772,-53.709,-179.651,6.643,149.116
C06805=1133.421,72.523,-53.692,-179.654,6.642,149.117
C06806=1133.425,72.274,-53.676,-179.657,6.640,149.117
C06807=1133.430,72.024,-53.659,-179.659,6.638,149.118
C06808=1133.436,71.775,-53.642,-179.662,6.638,149.118
C06809=1133.440,71.526,-53.625,-179.664,6.636,149.119
C06810=1133.444,71.276,-53.609,-179.668,6.635,149.119
C06811=1133.450,71.027,-53.592,-179.670,6.633,149.120
C06812=1133.455,70.777,-53.576,-179.672,6.632,149.120
C06813=1133.460,70.528,-53.560,-179.675,6.631,149.121
C06814=1133.465,70.279,-53.543,-179.678,6.629,149.121
C06815=1133.470,70.029,-53.526,-179.681,6.628,149.122
C06816=1133.475,69.780,-53.509,-179.683,6.627,149.122
C06817=1133.479,69.531,-53.493,-179.686,6.625,149.123
C06818=1133.485,69.280,-53.476,-179.689,6.624,149.123
C06819=1133.490,69.032,-53.460,-179.691,6.623,149.124
C06820=1133.495,68.782,-53.443,-179.694,6.621,149.124
C06821=1133.500,68.533,-53.427,-179.697,6.620,149.125
C06822=1133.504,68.283,-53.411,-179.700,6.618,149.125
C06823=1133.510,68.034,-53.394,-179.702,6.618,149.126
C06824=1133.515,67.785,-53.377,-179.705,6.616,149.126
C06825=1133.519,67.535,-53.361,-179.708,6.614,149.127
C06826=1133.525,67.286,-53.345,-179.710,6.614,149.127
C06827=1133.529,67.036,-53.328,-179.713,6.612,149.128
C06828=1133.535,66.787,-53.312,-179.716,6.611,149.128
C06829=1133.540,66.537,-53.296,-179.719,6.609,149.129
C06830=1133.545,66.288,-53.279,-179.721,6.608,149.129
C06831=1133.549,66.039,-53.263,-179.724,6.607,149.130
C06832=1133.555,65.789,-53.247,-179.727,6.605,149.130
C06833=1133.559,65.540,-53.230,-179.729,6.604,149.131
C06834=1133.564,65.291,-53.214,-179.732,6.603,149.131
C06835=1133.570,65.041,-53.198,-179.735,6.601,149.132
C06836=1133.574,64.791,-53.181,-179.737,6.601,149.132
C06837=1133.579,64.542,-53.165,-179.740,6.599,149.133
C06838=1133.584,64.292,-53.149,-179.743,6.597,149.133
C06839=1133.589,64.044,-53.132,-179.746,6.596,149.134
C06840=1133.594,63.793,-53.116,-179.748,6.595,149.134
C06841=1133.599,63.545,-53.100,-179.751,6.594,149.135
C06842=1133.604,63.295,-53.084,-179.754,6.592,149.135
C06843=1133.609,63.046,-53.068,-179.756,6.591,149.136
C06844=1133.614,62.796,-53.052,-179.759,6.590,149.136
C06845=1133.619,62.547,-53.036,-179.762,6.588,149.136
C06846=1133.624,62.297,-53.020,-179.764,6.587,149.137
C06847=1133.629,62.048,-53.003,-179.767,6.586,149.138
C06848=1133.634,61.799,-52.988,-179.770,6.584,149.138
C06849=1133.638,61.549,-52.971,-179.772,6.584,149.138
C06850=1133.644,61.300,-52.955,-179.775,6.582,149.139
C06851=1133.648,61.050,-52.939,-179.778,6.581,149.140
C06852=1133.654,60.801,-52.923,-179.780,6.580,149.140
C06853=1133.659,60.551,-52.906,-179.783,6.578,149.140
C06854=1133.664,60.302,-52.891,-179.786,6.577,149.141
C06855=1133.669,60.053,-52.875,-179.788,6.576,149.142
C06856=1133.673,59.803,-52.859,-179.791,6.574,149.142
C06857=1133.679,59.554,-52.843,-179.794,6.573,149.142
C06858=1133.683,59.304,-52.826,-179.796,6.572,149.143
C06859=1133.689,59.055,-52.811,-179.799,6.571,149.144
C06860=1133.694,58.806,-52.795,-179.802,6.569,149.144
C06861=1133.699,58.556,-52.779,-179.804,6.568,149.144
C06862=1133.704,58.306,-52.763,-179.807,6.567,149.145
C06863=1133.708,58.057,-52.746,-179.810,6.566,149.146
C06864=1133.714,57.808,-52.731,-179.812,6.565,149.146
C06865=1133.719,57.558,-52.715,-179.815,6.563,149.146
C06866=1133.724,57.309,-52.698,-179.817,6.562,149.147
C06867=1133.729,57.059,-52.683,-179.820,6.561,149.148
C06868=1133.734,56.809,-52.667,-179.823,6.559,149.148
C06869=1133.739,56.560,-52.651,-179.825,6.558,149.148
C06870=1133.744,56.311,-52.636,-179.829,6.557,149.149
C06871=1133.748,56.061,-52.620,-179.831,6.555,149.149
C06872=1133.754,55.812,-52.604,-179.834,6.555,149.150
C06873=1133.759,55.562,-52.588,-179.836,6.553,149.150
C06874=1133.764,55.313,-52.572,-179.839,6.552,149.151
C06875=1133.769,55.064,-52.556,-179.842,6.551,149.151
C06876=1133.774,54.814,-52.541,-179.844,6.549,149.152
C06877=1133.778,54.564,-52.525,-179.847,6.548,149.152
C06878=1133.783,54.316,-52.509,-179.850,6.547,149.153
C06879=1133.789,54.066,-52.493,-179.853,6.545,149.153
C06880=1133.794,53.816,-52.477,-179.855,6.545,149.154
C06881=1133.799,53.548,-52.460,-179.858,6.543,149.155
C06882=1133.805,53.279,-52.443,-179.861,6.542,149.155
C06883=1133.811,53.010,-52.427,-179.864,6.540,149.156
C06884=1133.815,52.742,-52.411,-179.866,6.540,149.156
C06885=1133.821,52.492,-52.395,-179.869,6.538,149.157
C06886=1133.825,52.243,-52.378,-179.872,6.537,149.157
C06887=1133.831,51.994,-52.363,-179.874,6.536,149.158
C06888=1133.835,51.744,-52.348,-179.877,6.534,149.158
C06889=1133.841,51.495,-52.332,-179.879,6.533,149.159
C06890=1133.846,51.245,-52.316,-179.883,6.532,149.159
C06891=1133.851,50.996,-52.301,-179.885,6.531,149.160
C06892=1133.856,50.746,-52.286,-179.887,6.530,149.160
C06893=1133.860,50.496,-52.270,-179.891,6.528,149.161
C06894=1133.866,50.247,-52.254,-179.893,6.528,149.161
C06895=1133.871,49.998,-52.239,-179.896,6.526,149.162
C06896=1133.876,49.748,-52.224,-179.898,6.525,149.162
C06897=1133.881,49.498,-52.208,-179.901,6.524,149.163
C06898=1133.886,49.249,-52.192,-179.904,6.522,149.163
C06899=1133.891,49.000,-52.177,-179.906,6.521,149.164
C06900=1133.896,48.750,-52.161,-179.909,6.520,149.164
C06901=1133.901,48.501,-52.146,-179.911,6.519,149.165
C06902=1133.905,48.251,-52.131,-179.914,6.518,149.165
C06903=1133.911,48.002,-52.115,-179.916,6.517,149.166
C06904=1133.916,47.752,-52.099,-179.919,6.516,149.166
C06905=1133.921,47.503,-52.084,-179.922,6.514,149.167
C06906=1133.926,47.254,-52.069,-179.924,6.513,149.167
C06907=1133.930,47.004,-52.053,-179.928,6.512,149.168
C06908=1133.936,46.754,-52.039,-179.930,6.511,149.168
C06909=1133.941,46.505,-52.023,-179.933,6.509,149.169
C06910=1133.946,46.256,-52.008,-179.935,6.509,149.170
C06911=1133.951,46.006,-51.992,-179.938,6.507,149.170
C06912=1133.955,45.756,-51.977,-179.941,6.506,149.170
C06913=1133.961,45.507,-51.961,-179.943,6.505,149.171
C06914=1133.966,45.258,-51.946,-179.946,6.504,149.172
C06915=1133.971,45.008,-51.932,-179.948,6.503,149.172
C06916=1133.977,44.759,-51.916,-179.951,6.501,149.172
C06917=1133.981,44.509,-51.901,-179.954,6.501,149.173
C06918=1133.987,44.260,-51.885,-179.956,6.499,149.174
C06919=1133.991,44.010,-51.870,-179.959,6.498,149.174
C06920=1133.996,43.760,-51.855,-179.961,6.497,149.174
C06921=1134.001,43.511,-51.840,-179.964,6.496,149.175
C06922=1134.006,43.262,-51.825,-179.967,6.495,149.176
C06923=1134.011,43.013,-51.810,-179.969,6.494,149.176
C06924=1134.017,42.763,-51.795,-179.972,6.493,149.177
C06925=1134.021,42.514,-51.780,-179.975,6.491,149.177
C06926=1134.027,42.264,-51.764,-179.977,6.490,149.178
C06927=1134.031,42.015,-51.749,-179.980,6.489,149.178
C06928=1134.036,41.764,-51.734,-179.983,6.488,149.179
C06929=1134.041,41.515,-51.719,-179.985,6.486,149.179
C06930=1134.047,41.266,-51.703,-179.988,6.486,149.180
C06931=1134.051,41.016,-51.689,-179.991,6.484,149.180
C06932=1134.057,40.767,-51.673,-179.993,6.483,149.181
C06933=1134.062,40.518,-51.658,-179.996,6.482,149.181
C06934=1134.067,40.268,-51.644,-179.998,6.481,149.182
C06935=1134.072,40.018,-51.629,179.999,6.480,149.182
C06936=1134.077,39.769,-51.613,179.997,6.479,149.183
C06937=1134.082,39.519,-51.599,179.994,6.478,149.183
C06938=1134.087,39.270,-51.584,179.991,6.477,149.184
C06939=1134.093,39.020,-51.569,179.989,6.475,149.184
C06940=1134.097,38.771,-51.554,179.986,6.475,149.185
C06941=1134.103,38.522,-51.538,179.983,6.473,149.185
C06942=1134.108,38.272,-51.524,179.981,6.472,149.186
C06943=1134.113,38.023,-51.508,179.978,6.471,149.186
C06944=1134.118,37.773,-51.494,179.976,6.470,149.187
C06945=1134.123,37.524,-51.479,179.973,6.469,149.187
C06946=1134.128,37.274,-51.464,179.971,6.468,149.188
C06947=1134.133,37.025,-51.449,179.967,6.467,149.189
C06948=1134.138,36.775,-51.435,179.965,6.466,149.189
C06949=1134.143,36.526,-51.419,179.963,6.464,149.189
C06950=1134.148,36.276,-51.405,179.960,6.464,149.190
C06951=1134.153,36.027,-51.390,179.957,6.462,149.191
C06952=1134.159,35.777,-51.375,179.955,6.461,149.191
C06953=1134.163,35.528,-51.360,179.952,6.460,149.192
C06954=1134.168,35.278,-51.346,179.950,6.459,149.192
C06955=1134.173,35.029,-51.330,179.947,6.458,149.193
C06956=1134.178,34.779,-51.316,179.944,6.457,149.193
C06957=1134.183,34.529,-51.302,179.942,6.456,149.194
C06958=1134.189,34.280,-51.286,179.939,6.455,149.194
C06959=1134.194,34.030,-51.272,179.937,6.454,149.195
C06960=1134.198,33.781,-51.257,179.934,6.453,149.195
C06961=1134.203,33.531,-51.243,179.932,6.452,149.196
C06962=1134.209,33.281,-51.228,179.929,6.450,149.196
C06963=1134.214,33.032,-51.213,179.926,6.450,149.197
C06964=1134.219,32.782,-51.199,179.923,6.448,149.197
C06965=1134.224,32.533,-51.184,179.921,6.447,149.198
C06966=1134.229,32.283,-51.169,179.918,6.446,149.199
C06967=1134.234,32.034,-51.154,179.916,6.445,149.199
C06968=1134.239,31.785,-51.141,179.913,6.444,149.199
C06969=1134.244,31.536,-51.126,179.910,6.443,149.200
C06970=1134.249,31.286,-51.111,179.908,6.442,149.201
C06971=1134.255,31.036,-51.096,179.906,6.441,149.201
C06972=1134.259,30.787,-51.081,179.903,6.440,149.202
C06973=1134.264,30.537,-51.067,179.900,6.439,149.202
C06974=1134.269,30.287,-51.053,179.898,6.438,149.203
C06975=1134.274,30.038,-51.039,179.895,6.437,149.203
C06976=1134.280,29.788,-51.023,179.893,6.436,149.204
C06977=1134.285,29.538,-51.009,179.890,6.434,149.204
C06978=1134.290,29.289,-50.995,179.887,6.434,149.205
C06979=1134.295,29.040,-50.981,179.885,6.433,149.205
C06980=1134.300,28.791,-50.966,179.882,6.431,149.206
C06981=1134.305,28.541,-50.951,179.880,6.431,149.206
C06982=1134.310,28.291,-50.937,179.877,6.429,149.207
C06983=1134.315,28.041,-50.922,179.875,6.428,149.207
C06984=1134.320,27.791,-50.908,179.871,6.427,149.208
C06985=1134.326,27.523,-50.892,179.869,6.426,149.208
C06986=1134.331,27.255,-50.877,179.866,6.425,149.209
C06987=1134.337,26.985,-50.862,179.864,6.424,149.210
C06988=1134.343,26.716,-50.845,179.860,6.423,149.210
C06989=1134.347,26.466,-50.831,179.858,6.422,149.211
C06990=1134.352,26.217,-50.817,179.856,6.421,149.211
C06991=1134.358,25.968,-50.803,179.853,6.420,149.212
C06992=1134.363,25.718,-50.789,179.850,6.419,149.212
C06993=1134.368,25.468,-50.774,179.848,6.418,149.213
C06994=1134.373,25.219,-50.760,179.845,6.417,149.213
C06995=1134.378,24.969,-50.746,179.843,6.416,149.214
C06996=1134.383,24.720,-50.732,179.840,6.415,149.214
C06997=1134.388,24.471,-50.717,179.837,6.414,149.215
C06998=1134.393,24.221,-50.703,179.835,6.413,149.216
C06999=1134.398,23.971,-50.688,179.833,6.412,149.216
C07000=1134.403,23.722,-50.674,179.830,6.411,149.217
C07001=1134.408,23.473,-50.660,179.827,6.410,149.217
C07002=1134.413,23.223,-50.646,179.825,6.408,149.218
C07003=1134.418,22.973,-50.632,179.822,6.408,149.218
C07004=1134.423,22.723,-50.617,179.820,6.407,149.219
C07005=1134.429,22.474,-50.604,179.817,6.405,149.219
C07006=1134.434,22.225,-50.589,179.814,6.405,149.220
C07007=1134.439,21.974,-50.576,179.812,6.403,149.220
C07008=1134.444,21.725,-50.561,179.809,6.403,149.221
C07009=1134.450,21.476,-50.547,179.807,6.402,149.221
C07010=1134.455,21.226,-50.533,179.804,6.401,149.222
C07011=1134.459,20.976,-50.519,179.802,6.400,149.222
C07012=1134.464,20.727,-50.505,179.799,6.399,149.223
C07013=1134.470,20.478,-50.491,179.796,6.398,149.223
C07014=1134.474,20.228,-50.477,179.794,6.397,149.224
C07015=1134.479,19.978,-50.463,179.791,6.396,149.225
C07016=1134.485,19.729,-50.449,179.789,6.395,149.225
C07017=1134.490,19.480,-50.435,179.787,6.394,149.226
C07018=1134.495,19.229,-50.421,179.783,6.393,149.226
C07019=1134.500,18.980,-50.407,179.781,6.392,149.227
C07020=1134.505,18.731,-50.393,179.779,6.391,149.227
C07021=1134.510,18.481,-50.379,179.776,6.390,149.228
C07022=1134.515,18.231,-50.364,179.774,6.389,149.228
C07023=1134.520,17.983,-50.351,179.771,6.388,149.229
C07024=1134.525,17.732,-50.337,179.768,6.387,149.229
C07025=1134.530,17.482,-50.323,179.766,6.386,149.230
C07026=1134.536,17.233,-50.309,179.764,6.385,149.230
C07027=1134.541,16.984,-50.295,179.761,6.384,149.231
C07028=1134.546,16.733,-50.281,179.758,6.383,149.231
C07029=1134.552,16.484,-50.267,179.756,6.383,149.232
C07030=1134.556,16.235,-50.254,179.753,6.381,149.233
C07031=1134.561,15.985,-50.240,179.751,6.381,149.233
C07032=1134.567,15.736,-50.226,179.748,6.379,149.234
C07033=1134.572,15.486,-50.212,179.745,6.379,149.234
C07034=1134.577,15.237,-50.198,179.743,6.378,149.235
C07035=1134.581,14.988,-50.184,179.740,6.376,149.235
C07036=1134.587,14.737,-50.171,179.738,6.376,149.236
C07037=1134.592,14.488,-50.157,179.736,6.375,149.236
C07038=1134.597,14.239,-50.143,179.733,6.373,149.237
C07039=1134.602,13.989,-50.130,179.730,6.373,149.237
C07040=1134.607,13.740,-50.116,179.728,6.372,149.238
C07041=1134.612,13.490,-50.102,179.726,6.371,149.238
C07042=1134.618,13.240,-50.088,179.723,6.370,149.239
C07043=1134.622,12.991,-50.075,179.720,6.369,149.240
C07044=1134.628,12.741,-50.061,179.718,6.368,149.240
C07045=1134.633,12.491,-50.047,179.715,6.367,149.241
C07046=1134.638,12.242,-50.033,179.713,6.366,149.241
C07047=1134.643,11.992,-50.020,179.711,6.365,149.242
C07048=1134.648,11.743,-50.006,179.707,6.364,149.242
C07049=1134.654,11.493,-49.993,179.705,6.363,149.243
C07050=1134.658,11.244,-49.979,179.703,6.363,149.243
C07051=1134.664,10.995,-49.965,179.700,6.361,149.244
C07052=1134.669,10.744,-49.952,179.698,6.361,149.244
C07053=1134.673,10.495,-49.938,179.695,6.360,149.245
C07054=1134.679,10.245,-49.925,179.692,6.359,149.245
C07055=1134.684,9.996,-49.911,179.690,6.358,149.246
C07056=1134.689,9.746,-49.898,179.688,6.357,149.246
C07057=1134.694,9.497,-49.884,179.685,6.357,149.247
C07058=1134.700,9.247,-49.870,179.682,6.355,149.248
C07059=1134.704,8.998,-49.857,179.680,6.354,149.248
C07060=1134.710,8.748,-49.844,179.678,6.354,149.249
C07061=1134.715,8.498,-49.829,179.675,6.352,149.249
C07062=1134.720,8.249,-49.817,179.672,6.352,149.250
C07063=1134.725,7.999,-49.802,179.670,6.351,149.250
C07064=1134.730,7.750,-49.790,179.668,6.350,149.251
C07065=1134.736,7.500,-49.776,179.665,6.349,149.251
C07066=1134.741,7.251,-49.762,179.662,6.348,149.252
C07067=1134.746,7.000,-49.749,179.660,6.347,149.252
C07068=1134.751,6.751,-49.735,179.657,6.346,149.253
C07069=1134.756,6.501,-49.723,179.655,6.345,149.254
C07070=1134.762,6.252,-49.709,179.653,6.344,149.254
C07071=1134.766,6.002,-49.696,179.650,6.344,149.255
C07072=1134.772,5.753,-49.682,179.647,6.342,149.255
C07073=1134.776,5.503,-49.669,179.645,6.342,149.256
C07074=1134.782,5.254,-49.656,179.642,6.341,149.256
C07075=1134.787,5.003,-49.642,179.640,6.340,149.257
C07076=1134.792,4.755,-49.629,179.637,6.339,149.257
C07077=1134.798,4.505,-49.615,179.635,6.338,149.258
C07078=1134.802,4.255,-49.603,179.633,6.338,149.258
C07079=1134.808,4.006,-49.589,179.630,6.337,149.259
C07080=1134.812,3.756,-49.576,179.627,6.335,149.260
C07081=1134.818,3.506,-49.562,179.625,6.335,149.260
C07082=1134.823,3.256,-49.549,179.623,6.334,149.260
C07083=1134.828,3.007,-49.536,179.620,6.333,149.261
C07084=1134.833,2.757,-49.523,179.617,6.332,149.262
C07085=1134.839,2.508,-49.509,179.615,6.331,149.262
C07086=1134.844,2.258,-49.497,179.613,6.331,149.263
C07087=1134.848,2.009,-49.483,179.610,6.330,149.263
C07088=1134.854,1.759,-49.470,179.608,6.328,149.264
C07089=1134.860,1.489,-49.456,179.605,6.328,149.264
C07090=1134.864,1.220,-49.441,179.602,6.326,149.265
C07091=1134.871,0.951,-49.427,179.599,6.326,149.266
C07092=1134.876,0.681,-49.413,179.597,6.325,149.266
C07093=1134.881,0.432,-49.400,179.594,6.324,149.267
C07094=1134.886,0.182,-49.387,179.592,6.323,149.267
C07095=1134.892,-0.067,-49.374,179.589,6.323,149.268
C07096=1134.897,-0.317,-49.361,179.587,6.322,149.268
C07097=1134.902,-0.567,-49.347,179.584,6.320,149.269
C07098=1134.907,-0.816,-49.335,179.582,6.320,149.269
C07099=1134.912,-1.066,-49.322,179.579,6.319,149.270
C07100=1134.917,-1.315,-49.308,179.577,6.318,149.270
C07101=1134.922,-1.565,-49.295,179.575,6.318,149.271
C07102=1134.927,-1.815,-49.282,179.572,6.316,149.272
C07103=1134.933,-2.064,-49.269,179.570,6.315,149.272
C07104=1134.938,-2.314,-49.257,179.567,6.315,149.273
C07105=1134.943,-2.564,-49.243,179.565,6.314,149.273
C07106=1134.948,-2.813,-49.230,179.562,6.313,149.274
C07107=1134.953,-3.063,-49.218,179.559,6.312,149.274
C07108=1134.959,-3.313,-49.204,179.557,6.311,149.275
C07109=1134.964,-3.562,-49.192,179.555,6.310,149.275
C07110=1134.969,-3.812,-49.179,179.552,6.310,149.276
C07111=1134.975,-4.061,-49.166,179.550,6.308,149.276
C07112=1134.979,-4.311,-49.153,179.547,6.308,149.277
C07113=1134.984,-4.561,-49.140,179.545,6.307,149.278
C07114=1134.989,-4.810,-49.128,179.543,6.306,149.278
C07115=1134.995,-5.060,-49.114,179.540,6.306,149.279
C07116=1135.000,-5.310,-49.102,179.537,6.304,149.279
C07117=1135.005,-5.559,-49.089,179.535,6.304,149.280
C07118=1135.010,-5.809,-49.075,179.533,6.303,149.280
C07119=1135.015,-6.059,-49.063,179.530,6.302,149.281
C07120=1135.020,-6.308,-49.050,179.528,6.302,149.281
C07121=1135.026,-6.557,-49.038,179.525,6.300,149.282
C07122=1135.031,-6.808,-49.024,179.522,6.300,149.282
C07123=1135.036,-7.057,-49.011,179.520,6.299,149.283
C07124=1135.041,-7.306,-48.999,179.518,6.298,149.284
C07125=1135.046,-7.555,-48.986,179.515,6.298,149.284
C07126=1135.051,-7.805,-48.973,179.513,6.297,149.285
C07127=1135.057,-8.055,-48.960,179.510,6.296,149.285
C07128=1135.062,-8.305,-48.948,179.508,6.295,149.286
C07129=1135.067,-8.554,-48.936,179.506,6.294,149.286
C07130=1135.072,-8.804,-48.923,179.503,6.294,149.287
C07131=1135.077,-9.054,-48.910,179.501,6.293,149.287
C07132=1135.083,-9.303,-48.897,179.499,6.292,149.288
C07133=1135.088,-9.553,-48.884,179.495,6.291,149.289
C07134=1135.093,-9.802,-48.872,179.493,6.290,149.289
C07135=1135.098,-10.053,-48.859,179.491,6.289,149.289
C07136=1135.103,-10.302,-48.847,179.488,6.289,149.290
C07137=1135.108,-10.551,-48.834,179.486,6.288,149.291
C07138=1135.114,-10.801,-48.821,179.484,6.287,149.291
C07139=1135.119,-11.050,-48.808,179.481,6.286,149.292
C07140=1135.124,-11.301,-48.796,179.479,6.285,149.292
C07141=1135.129,-11.550,-48.783,179.476,6.284,149.293
C07142=1135.134,-11.799,-48.771,179.474,6.284,149.293
C07143=1135.139,-12.049,-48.758,179.472,6.283,149.294
C07144=1135.144,-12.298,-48.746,179.469,6.282,149.294
C07145=1135.149,-12.549,-48.733,179.466,6.281,149.295
C07146=1135.155,-12.798,-48.720,179.464,6.280,149.296
C07147=1135.160,-13.048,-48.708,179.462,6.280,149.296
C07148=1135.166,-13.298,-48.696,179.459,6.279,149.297
C07149=1135.171,-13.547,-48.683,179.457,6.278,149.297
C07150=1135.176,-13.796,-48.671,179.455,6.278,149.298
C07151=1135.180,-14.046,-48.658,179.452,6.277,149.298
C07152=1135.186,-14.296,-48.646,179.449,6.276,149.299
C07153=1135.191,-14.546,-48.633,179.447,6.275,149.299
C07154=1135.196,-14.795,-48.621,179.444,6.274,149.300
C07155=1135.201,-15.045,-48.609,179.442,6.274,149.300
C07156=1135.207,-15.294,-48.596,179.440,6.273,149.301
C07157=1135.212,-15.544,-48.584,179.437,6.272,149.302
C07158=1135.217,-15.793,-48.572,179.435,6.272,149.302
C07159=1135.222,-16.043,-48.559,179.433,6.271,149.303
C07160=1135.227,-16.293,-48.547,179.430,6.270,149.303
C07161=1135.232,-16.543,-48.534,179.428,6.269,149.304
C07162=1135.237,-16.792,-48.521,179.425,6.268,149.304
C07163=1135.243,-17.042,-48.510,179.423,6.268,149.305
C07164=1135.248,-17.291,-48.497,179.421,6.267,149.305
C07165=1135.253,-17.541,-48.485,179.418,6.266,149.306
C07166=1135.258,-17.790,-48.473,179.416,6.266,149.306
C07167=1135.264,-18.040,-48.461,179.414,6.265,149.307
C07168=1135.269,-18.290,-48.448,179.411,6.264,149.307
C07169=1135.273,-18.540,-48.435,179.408,6.263,149.308
C07170=1135.279,-18.790,-48.423,179.406,6.262,149.309
C07171=1135.284,-19.039,-48.411,179.404,6.261,149.309
C07172=1135.289,-19.289,-48.399,179.401,6.261,149.310
C07173=1135.295,-19.538,-48.386,179.399,6.260,149.310
C07174=1135.300,-19.788,-48.374,179.397,6.259,149.311
C07175=1135.305,-20.037,-48.362,179.394,6.259,149.311
C07176=1135.311,-20.287,-48.350,179.392,6.258,149.312
C07177=1135.316,-20.537,-48.337,179.390,6.257,149.312
C07178=1135.321,-20.787,-48.325,179.386,6.256,149.313
C07179=1135.327,-21.037,-48.313,179.384,6.255,149.313
C07180=1135.331,-21.286,-48.301,179.382,6.255,149.314
C07181=1135.336,-21.536,-48.289,179.379,6.254,149.315
C07182=1135.341,-21.785,-48.277,179.377,6.253,149.315
C07183=1135.347,-22.035,-48.265,179.375,6.253,149.316
C07184=1135.352,-22.284,-48.252,179.372,6.252,149.316
C07185=1135.357,-22.534,-48.240,179.370,6.251,149.317
C07186=1135.363,-22.784,-48.229,179.368,6.251,149.317
C07187=1135.368,-23.033,-48.216,179.365,6.250,149.318
C07188=1135.373,-23.283,-48.204,179.363,6.249,149.318
C07189=1135.378,-23.532,-48.192,179.361,6.249,149.319
C07190=1135.383,-23.782,-48.180,179.358,6.247,149.320
C07191=1135.389,-24.032,-48.168,179.355,6.247,149.320
C07192=1135.394,-24.281,-48.156,179.353,6.246,149.321
C07193=1135.399,-24.552,-48.143,179.351,6.245,149.321
C07194=1135.405,-24.821,-48.130,179.348,6.245,149.322
C07195=1135.410,-25.092,-48.117,179.346,6.244,149.322
C07196=1135.416,-25.362,-48.104,179.343,6.243,149.323
C07197=1135.422,-25.611,-48.093,179.340,6.242,149.324
C07198=1135.427,-25.861,-48.080,179.338,6.241,149.324
C07199=1135.432,-26.111,-48.068,179.336,6.241,149.325
C07200=1135.438,-26.361,-48.056,179.333,6.240,149.325
C07201=1135.443,-26.611,-48.044,179.331,6.240,149.326
C07202=1135.447,-26.860,-48.032,179.329,6.239,149.326
C07203=1135.453,-27.109,-48.021,179.326,6.238,149.327
C07204=1135.458,-27.359,-48.009,179.324,6.238,149.327
C07205=1135.464,-27.609,-47.997,179.322,6.237,149.328
C07206=1135.468,-27.858,-47.985,179.319,6.236,149.329
C07207=1135.474,-28.108,-47.973,179.317,6.236,149.329
C07208=1135.479,-28.358,-47.961,179.315,6.235,149.329
C07209=1135.484,-28.608,-47.950,179.312,6.234,149.330
C07210=1135.489,-28.857,-47.937,179.310,6.234,149.331
C07211=1135.494,-29.107,-47.925,179.308,6.233,149.331
C07212=1135.500,-29.357,-47.913,179.305,6.232,149.332
C07213=1135.505,-29.606,-47.902,179.303,6.232,149.332
C07214=1135.510,-29.856,-47.891,179.300,6.230,149.333
C07215=1135.516,-30.106,-47.879,179.298,6.230,149.333
C07216=1135.520,-30.355,-47.867,179.295,6.229,149.334
C07217=1135.526,-30.605,-47.855,179.293,6.228,149.334
C07218=1135.531,-30.855,-47.843,179.291,6.228,149.335
C07219=1135.536,-31.104,-47.832,179.288,6.227,149.336
C07220=1135.541,-31.354,-47.820,179.286,6.226,149.336
C07221=1135.547,-31.604,-47.808,179.284,6.225,149.337
C07222=1135.552,-31.853,-47.797,179.281,6.225,149.337
C07223=1135.557,-32.103,-47.785,179.279,6.224,149.338
C07224=1135.562,-32.352,-47.772,179.277,6.223,149.338
C07225=1135.567,-32.602,-47.761,179.274,6.223,149.339
C07226=1135.573,-32.852,-47.749,179.272,6.222,149.339
C07227=1135.578,-33.102,-47.737,179.270,6.221,149.340
C07228=1135.583,-33.352,-47.726,179.267,6.221,149.341
C07229=1135.589,-33.601,-47.715,179.265,6.220,149.341
C07230=1135.593,-33.850,-47.703,179.263,6.219,149.341
C07231=1135.599,-34.100,-47.691,179.260,6.219,149.342
C07232=1135.604,-34.350,-47.679,179.258,6.218,149.343
C07233=1135.609,-34.600,-47.668,179.256,6.217,149.343
C07234=1135.614,-34.850,-47.656,179.253,6.217,149.344
C07235=1135.620,-35.099,-47.645,179.251,6.216,149.344
C07236=1135.625,-35.349,-47.634,179.249,6.216,149.345
C07237=1135.631,-35.599,-47.622,179.247,6.215,149.345
C07238=1135.635,-35.848,-47.610,179.244,6.214,149.346
C07239=1135.641,-36.098,-47.598,179.242,6.214,149.346
C07240=1135.646,-36.347,-47.588,179.240,6.213,149.347
C07241=1135.651,-36.597,-47.576,179.237,6.212,149.348
C07242=1135.656,-36.847,-47.564,179.235,6.212,149.348
C07243=1135.662,-37.097,-47.552,179.233,6.211,149.349
C07244=1135.668,-37.346,-47.541,179.230,6.210,149.349
C07245=1135.672,-37.595,-47.530,179.228,6.210,149.350
C07246=1135.678,-37.846,-47.518,179.225,6.209,149.350
C07247=1135.683,-38.096,-47.507,179.223,6.208,149.351
C07248=1135.688,-38.346,-47.495,179.221,6.208,149.351
C07249=1135.693,-38.594,-47.484,179.218,6.207,149.352
C07250=1135.699,-38.844,-47.473,179.216,6.206,149.352
C07251=1135.704,-39.094,-47.461,179.214,6.206,149.353
C07252=1135.709,-39.344,-47.449,179.211,6.205,149.353
C07253=1135.714,-39.593,-47.438,179.209,6.204,149.354
C07254=1135.720,-39.843,-47.427,179.207,6.204,149.355
C07255=1135.725,-40.093,-47.416,179.204,6.203,149.355
C07256=1135.731,-40.342,-47.404,179.202,6.202,149.356
C07257=1135.735,-40.592,-47.393,179.199,6.202,149.356
C07258=1135.740,-40.842,-47.382,179.197,6.201,149.357
C07259=1135.746,-41.092,-47.370,179.195,6.200,149.357
C07260=1135.751,-41.341,-47.360,179.192,6.200,149.358
C07261=1135.757,-41.591,-47.348,179.190,6.199,149.358
C07262=1135.761,-41.841,-47.337,179.188,6.198,149.359
C07263=1135.767,-42.091,-47.325,179.186,6.198,149.359
C07264=1135.772,-42.339,-47.314,179.184,6.198,149.360
C07265=1135.778,-42.590,-47.303,179.182,6.197,149.361
C07266=1135.782,-42.840,-47.291,179.179,6.196,149.361
